Yaskawa INFORM job: X2_8A-21A(90,0)_HARDOX.JBI

/JOB
//NAME X2_8A-21A(90,0)_HARDOX
///FOLDERNAME X2
//POS
///NPOS 1752,1752,1752,46,0,0
///TOOL 0
///POSTYPE PULSE
///PULSE
C00000=-12667,-135547,-130714,31270,45596,0
C00001=-9315,-159766,-119262,-3212,6219,55552
C00002=-157761,-135547,-130714,31270,45596,-69143
C00003=-154472,-113934,-104337,41712,51336,-70449
C00004=-149832,-108771,-100172,39130,49259,-68869
C00005=-148058,-106656,-98467,38074,48499,-68236
C00006=-148062,-106275,-96666,38578,47777,-68578
C00007=-148058,-106656,-98467,38074,48499,-68236
C00008=-147997,-106381,-96958,38469,47847,-68508
C00009=-145894,-104035,-96109,36815,47477,-67498
C00010=-147997,-106381,-96958,38469,47847,-68508
C00011=-154410,-113635,-102825,42095,50721,-70729
C00012=-154342,-120637,-107041,25827,48602,-38771
C00013=-150292,-111683,-102360,22573,48994,-36710
C00014=-148798,-108210,-100464,21373,49171,-35962
C00015=-146664,-105787,-99597,19708,49308,-34937
C00016=-146949,-106220,-99797,19932,49282,-35074
C00017=-147721,-103636,-97533,20478,49410,-35405
C00018=-146949,-106220,-99797,19932,49282,-35074
C00019=-152261,-118724,-106469,24248,48548,-37770
C00020=-148295,-114597,-117137,-6490,60568,-69086
C00021=-147868,-109631,-111600,-6790,59752,-68875
C00022=-147704,-107727,-109395,-6911,59390,-68790
C00023=-147708,-107860,-107783,-6984,58336,-68724
C00024=-147704,-107727,-109395,-6911,59390,-68790
C00025=-147723,-107760,-107968,-6963,58499,-68740
C00026=-147306,-102596,-106094,-7098,60024,-68678
C00027=-147723,-107760,-107968,-6963,58499,-68740
C00028=-148315,-114751,-115749,-6537,59639,-69038
C00029=-148355,-114889,-117236,-6461,60467,-69101
C00030=-147925,-109892,-111692,-6763,59663,-68890
C00031=-147761,-107977,-109485,-6884,59305,-68805
C00032=-147764,-108104,-107870,-6957,58254,-68739
C00033=-147777,-108153,-108078,-6942,58354,-68751
C00034=-147358,-102980,-106206,-7078,59886,-68688
C00035=-147777,-108153,-108078,-6942,58354,-68751
C00036=-148373,-115211,-115873,-6515,59468,-69049
C00037=-147696,-122269,-111871,-35505,39043,-51945
C00038=-147690,-118447,-100224,-39719,34874,-49579
C00039=-148491,-109409,-94254,-38171,35277,-50420
C00040=-148787,-105724,-91002,-38010,35060,-50504
C00041=-148789,-105382,-89977,-38411,34697,-50285
C00042=-149058,-101689,-89016,-37046,35623,-51030
C00043=-149145,-100783,-88679,-36755,35795,-51189
C00044=-149058,-101689,-89016,-37046,35623,-51030
C00045=-145777,-99657,-88811,-39022,37803,-49998
C00046=-148139,-100407,-89095,-37251,36591,-50936
C00047=-145777,-99657,-88811,-39022,37803,-49998
C00048=-147690,-118447,-100224,-39719,34874,-49579
C00049=-128033,-128545,-103748,-39689,32513,-43973
C00050=-128383,-118409,-97778,-37905,33566,-44930
C00051=-128511,-114277,-94563,-37658,33626,-45064
C00052=-128512,-113804,-93446,-38069,33271,-44843
C00053=-129119,-111006,-93029,-36452,33958,-45715
C00054=-129434,-109852,-92636,-35862,34111,-46033
C00055=-128358,-113721,-93936,-37885,33613,-44941
C00056=-176216,-70111,-78093,55162,70856,-80763
C00057=-174311,-70781,-78417,54616,69674,-80426
C00058=-176216,-70111,-78093,55162,70856,-80763
C00059=-181747,-69996,-81392,56304,75271,-81045
C00060=-178033,-77165,-93769,42680,75059,-77098
C00061=-164745,-109340,-116699,-3009,62053,-68278
C00062=-145851,-112599,-102075,-47717,41998,-56322
C00063=-148044,-104803,-96379,-45883,41204,-57334
C00064=-148864,-101708,-93474,-45490,40644,-57533
C00065=-148866,-101457,-92299,-45986,40221,-57239
C00066=-148863,-101834,-94104,-45225,40876,-57690
C00067=-145127,-99228,-91361,-47944,42572,-56214
C00068=-147466,-100038,-91670,-46636,41186,-56907
C00069=-145127,-99228,-91361,-47944,42572,-56214
C00070=-146129,-107372,-95667,-48598,40993,-55782
C00071=-148216,-109089,-93488,-49289,38371,-55335
C00072=-148344,-107837,-93052,-48851,38553,-55585
C00073=-147906,-112054,-94498,-50363,37947,-54724
C00074=-145851,-112599,-102075,-47717,41998,-56322
C00075=-158250,-140903,-124067,-47621,67451,-49320
C00076=-161740,-133075,-117656,-46661,65672,-50232
C00077=-162335,-130592,-114553,-46699,64919,-50156
C00078=-162276,-129951,-113381,-46845,64676,-49998
C00079=-160420,-132544,-115533,-47350,65644,-49520
C00080=-135901,-74424,-73697,-74364,100921,-31256
C00081=-137788,-75503,-74147,-74218,99532,-31324
C00082=-138769,-76027,-74362,-74146,98812,-31363
C00083=-135901,-74424,-73697,-74364,100921,-31256
C00084=-149282,-147643,-98518,-79858,51263,-26133
C00085=-149394,-146891,-98381,-79629,51249,-26315
C00086=-148448,-152811,-99407,-81432,51428,-24854
C00087=-139735,-166147,-105854,-82069,56849,-22658
C00088=-180438,-97574,-115199,-33764,102267,52414
C00089=-189965,-108899,-115705,-31971,94091,51156
C00090=-189186,-107218,-114531,-32087,94499,51341
C00091=-189186,-107583,-113435,-32037,93763,51550
C00092=-190629,-109833,-115910,-31859,93547,51055
C00093=-186867,-102382,-113240,-32521,96788,51574
C00094=-187005,-102964,-110979,-32373,95300,51952
C00095=-188888,-106610,-112304,-32065,93703,51681
C00096=-187005,-102964,-110979,-32373,95300,51952
C00097=-188021,-107681,-112675,-32159,93748,52003
C00098=-189590,-103281,-111094,-32025,94271,51250
C00099=-188021,-107681,-112675,-32159,93748,52003
C00100=-180438,-97574,-115199,-33764,102267,52414
C00101=-185735,-83978,-109774,-33564,103394,50026
C00102=-199988,-77820,-108712,11582,98175,-38155
C00103=-204749,-56978,-92496,29836,109182,-47433
C00104=-202460,-56662,-91339,29422,107990,-46925
C00105=-201413,-57385,-91726,29256,107546,-46663
C00106=-201611,-57041,-91542,29296,107663,-46703
C00107=-201611,-58240,-90431,29070,106521,-47008
C00108=-203359,-50274,-87822,29763,109247,-46906
C00109=-195470,-25798,-72981,29209,109868,-43903
C00110=-195013,-27562,-73704,29036,109327,-43888
C00111=-194283,-28250,-74172,28893,109053,-43704
C00112=-194480,-28066,-74047,28932,109127,-43754
C00113=-194480,-29296,-73135,28708,108075,-44034
C00114=-195605,-24849,-71507,29147,109538,-44038
C00115=-191110,-5546,-57842,28597,109561,-42465
C00116=-192519,-3768,-54500,33008,111368,-41387
C00117=-191992,-5303,-55742,32912,111174,-41254
C00118=-192059,-5108,-55586,32924,111198,-41271
C00119=-192059,-6294,-54683,32651,110210,-41583
C00120=-192882,-2296,-53893,33162,111810,-41382
C00121=-203365,-15491,-64400,34648,115083,-44256
C00122=-218411,-26661,-75493,58573,107247,-46176
C00123=-145332,-87800,-123084,4045,108310,15756
C00124=-109199,-104290,-129101,-21867,105305,43874
C00125=-112610,-115777,-129409,-14908,94573,36374
C00126=-117115,-112620,-124614,-14006,92529,35127
C00127=-118008,-112320,-123068,-13816,91609,34934
C00128=-118007,-112900,-122267,-13806,90840,35020
C00129=-118044,-112536,-122505,-13803,91159,34973
C00130=-118576,-105776,-120168,-13731,93052,34586
C00131=-118044,-112536,-122505,-13803,91159,34973
C00132=-125955,-111499,-122045,-12179,90192,32457
C00133=-127333,-111877,-122174,-11884,89885,32033
C00134=-124755,-111115,-121914,-12435,90480,32824
C00135=-119624,-116552,-128230,-13509,92325,34321
C00136=-117231,-121833,-124467,-22052,85463,28755
C00137=-122341,-114124,-118662,-20866,84531,27121
C00138=-123318,-113111,-117155,-20643,83910,26885
C00139=-123641,-113323,-116249,-20585,83205,26892
C00140=-123595,-112804,-116375,-20585,83540,26851
C00141=-123397,-106736,-114247,-20589,85286,26623
C00142=-123595,-112804,-116375,-20585,83540,26851
C00143=-116023,-114044,-115764,-22346,84523,29358
C00144=-117346,-116777,-115957,-22098,82979,29171
C00145=-118867,-116723,-116143,-21757,82713,28674
C00146=-116293,-116772,-115815,-22329,83179,29512
C00147=-117231,-121833,-124467,-22052,85463,28755
C00148=-154726,-134692,-133300,19029,79240,32627
C00149=-155157,-123239,-125350,19102,80279,32639
C00150=-155214,-122106,-123677,19140,79867,32554
C00151=-155216,-122330,-122794,19175,79245,32454
C00152=-155272,-122641,-123186,19186,79334,32449
C00153=-154565,-115790,-120970,18882,81218,32994
C00154=-155272,-122449,-123985,19155,79894,32538
C00155=-110972,-119209,-121408,-15853,79302,48266
C00156=-109086,-133769,-122042,-16854,72857,49812
C00157=-111848,-135958,-122676,-16103,71595,48979
C00158=-109086,-133769,-122042,-16854,72857,49812
C00159=-108592,-130707,-130810,-16554,79646,49045
C00160=-120610,-122471,-119242,-21572,81234,22537
C00161=-120610,-122484,-118172,-21604,80613,22649
C00162=-120610,-122391,-116483,-21658,79689,22817
C00163=-120610,-122419,-116833,-21647,79876,22783
C00164=-120610,-122423,-116832,-21647,79874,22783
C00165=-120610,-122419,-116833,-21647,79876,22783
C00166=-120610,-122416,-116761,-21649,79836,22790
C00167=-120610,-122436,-116768,-21650,79830,22791
C00168=-120610,-122416,-116761,-21649,79836,22790
C00169=-120611,-122370,-120508,-21535,82009,22397
C00170=-120611,-120494,-126735,-3133,87635,4471
C00171=-120611,-121772,-123926,-3138,85252,4531
C00172=-120611,-122092,-122744,-3141,84362,4553
C00173=-120611,-122362,-121169,-3146,83256,4581
C00174=-120611,-122286,-121724,-3144,83636,4571
C00175=-120611,-122290,-121724,-3144,83633,4571
C00176=-120611,-122286,-121724,-3144,83636,4571
C00177=-120611,-121006,-125813,-3134,86805,4492
C00178=-120621,-120378,-125991,-12397,109990,35253
C00179=-136832,-143297,-133894,-19017,104291,40845
C00180=-187686,-122249,-118318,-34521,102174,42234
C00181=-187703,-122088,-115580,-34298,100833,42653
C00182=-187707,-122010,-114917,-34250,100525,42749
C00183=-187713,-121734,-113169,-34135,99743,42991
C00184=-187707,-122010,-114917,-34250,100525,42749
C00185=-187770,-121697,-112491,-32279,113674,44764
C00186=-187767,-121692,-112491,-32279,113678,44765
C00187=-187770,-121697,-112491,-32279,113674,44764
C00188=-187667,-121438,-112064,-34928,84963,41689
C00189=-187673,-121448,-112068,-34927,84958,41688
C00190=-187667,-121438,-112064,-34928,84963,41689
C00191=-187641,-121957,-115421,-34884,86463,41227
C00192=-173591,-141106,-131528,-9997,106250,69327
C00193=-160878,-120510,-126471,-37,121976,81968
C00194=-160881,-121699,-123664,-37,119637,81967
C00195=-160883,-121991,-122485,-37,118762,81967
C00196=-160886,-122244,-120905,-37,117660,81966
C00197=-160884,-122111,-121864,-37,118318,81967
C00198=-160882,-122100,-121862,-36,118322,81968
C00199=-160884,-122111,-121864,-37,118318,81967
C00200=-160879,-120821,-125908,-37,121469,81968
C00201=-160879,-120821,-131564,-37,121469,81968
C00202=-166129,-114439,-129167,13521,133132,-54375
C00203=-82387,-124374,-130385,21792,102809,-55833
C00204=-37550,-124758,-124791,27166,84975,-54517
C00205=-35933,-124831,-122904,26864,83389,-54284
C00206=-35589,-124875,-121597,26827,82538,-54351
C00207=-35584,-124889,-121174,26839,82296,-54405
C00208=-35764,-126387,-121953,26892,82093,-54519
C00209=-31633,-125451,-121673,25972,81076,-53208
C00210=-35764,-126387,-121953,26892,82093,-54519
C00211=-46981,-157328,-126723,35790,81436,-33730
C00212=-42905,-153934,-122174,35701,78867,-32870
C00213=-42758,-143813,-119569,35389,81762,-31868
C00214=-42905,-153934,-122174,35701,78867,-32870
C00215=-53188,-117519,-120731,36414,97747,-30962
C00216=-95179,-109851,-129540,3422,106316,17944
C00217=-143691,-100776,-119079,-26047,122130,73021
C00218=-146029,-112499,-120098,-24937,116556,73463
C00219=-147204,-116618,-119576,-24569,113992,73590
C00220=-147487,-116577,-118677,-24502,113425,73607
C00221=-146967,-116625,-120319,-24630,114475,73574
C00222=-147345,-121113,-121824,-24401,113105,73737
C00223=-146899,-128254,-123879,-23878,111030,74376
C00224=-147345,-121113,-121824,-24401,113105,73737
C00225=-118081,-135478,-120686,-30293,109901,65237
C00226=-118366,-136707,-118609,-29972,108136,65614
C00227=-120887,-140213,-119894,-30302,106351,65070
C00228=-118366,-136707,-118609,-29972,108136,65614
C00229=-117820,-130449,-123242,-31209,113594,64262
C00230=-93926,-103398,-125362,-18301,106221,39936
C00231=-72688,-110808,-124077,-7134,85250,24096
C00232=-75848,-101444,-116923,-6191,85411,23073
C00233=-76170,-100985,-115528,-6097,84767,23002
C00234=-76167,-101481,-114835,-6104,84090,23035
C00235=-78739,-96930,-113773,-5320,85595,22140
C00236=-79843,-95445,-113201,-4985,85938,21775
C00237=-77748,-98228,-114268,-5620,85298,22470
C00238=-140085,-104632,-109249,40944,98797,-6712
C00239=-140263,-103640,-106572,40817,98007,-7102
C00240=-137942,-102173,-106029,40697,97269,-6378
C00241=-140263,-103640,-106572,40817,98007,-7102
C00242=-135988,-101428,-112112,41019,99549,-4631
C00243=-141957,-83285,-117139,12315,91699,6710
C00244=-161957,-129781,-122866,-20018,67926,12328
C00245=-166016,-109699,-113650,-17211,72980,10098
C00246=-166795,-105246,-111748,-16434,74862,9605
C00247=-165677,-113012,-111900,-18316,68836,10778
C00248=-162725,-116093,-113629,-19548,69016,11850
C00249=-162651,-107484,-110669,-19284,71494,11460
C00250=-162725,-116093,-113629,-19548,69016,11850
C00251=-155151,-112727,-112486,-22270,71877,14160
C00252=-155120,-113819,-110277,-22518,70103,14518
C00253=-159000,-114269,-110433,-21107,68960,13264
C00254=-155120,-113819,-110277,-22518,70103,14518
C00255=-155137,-138999,-124748,-23105,66364,15269
C00256=-81055,-115973,-127517,23586,109336,-64560
C00257=-76492,-127739,-126040,22738,101683,-64421
C00258=-76072,-128597,-125529,22671,100870,-64425
C00259=-76065,-128640,-125326,22657,100732,-64448
C00260=-76072,-128576,-125785,22685,101025,-64394
C00261=-82641,-146978,-130130,22016,96499,-67668
C00262=-81130,-155003,-132256,21951,93476,-67670
C00263=-82641,-146978,-130130,22016,96499,-67668
C00264=-84000,-144678,-127518,21929,96467,-68175
C00265=-84000,-143983,-126065,21900,95967,-68269
C00266=-83327,-146231,-127404,21916,95478,-68108
C00267=-88356,-135439,-132684,22407,104994,-68175
C00268=-104080,-128245,-132212,-31995,84146,-22143
C00269=-106783,-105266,-117364,-31197,85468,-23533
C00270=-107129,-103609,-115494,-31111,85090,-23558
C00271=-107127,-104217,-114421,-31144,84251,-23329
C00272=-107044,-104571,-114816,-31164,84333,-23320
C00273=-107880,-99055,-112779,-30885,85404,-23924
C00274=-107044,-104571,-114816,-31164,84333,-23320
C00275=-105114,-115284,-123193,-31689,84721,-22698
C00276=-105208,-113465,-123990,-31624,85910,-23065
C00277=-106823,-104635,-117017,-31184,85549,-23570
C00278=-107122,-103295,-115264,-31113,85109,-23561
C00279=-107121,-103855,-114286,-31142,84342,-23351
C00280=-107087,-104437,-114776,-31151,84356,-23343
C00281=-107921,-98925,-112738,-30873,85426,-23945
C00282=-107087,-104437,-114776,-31151,84356,-23343
C00283=-105701,-116384,-125830,-31502,85418,-23114
C00284=-79137,-116524,-127291,-7118,77084,38210
C00285=-66518,-158449,-133200,-8588,59166,50817
C00286=-70166,-147728,-127011,-6864,60501,49298
C00287=-71549,-143558,-123868,-6244,60595,48757
C00288=-71544,-142942,-122687,-6271,60188,48782
C00289=-71412,-140542,-122600,-6259,61371,48766
C00290=-74130,-137647,-121783,-5023,62161,47690
C00291=-71412,-140542,-122600,-6259,61371,48766
C00292=-59221,-85077,-106862,-19044,97138,55247
C00293=-59772,-90133,-108950,-18878,95774,55276
C00294=-59221,-85077,-106862,-19044,97138,55247
C00295=-65406,-128676,-128270,-8670,80773,42177
C00296=-57064,-112054,-129147,-2862,108793,29097
C00297=-70948,-123089,-127271,10962,111372,-380
C00298=-67644,-116564,-123033,11394,111660,848
C00299=-67644,-116773,-122597,11361,111292,811
C00300=-67644,-116291,-123546,11437,112109,893
C00301=-70770,-123262,-125779,10903,110357,-412
C00302=-70770,-123588,-124717,10837,109552,-488
C00303=-69306,-120453,-123728,11077,110342,115
C00304=-70770,-123283,-125719,10898,110311,-416
C00305=-70770,-119886,-130778,11344,115083,53
C00306=-68413,-122856,-123349,22437,117236,58
C00307=-67404,-122631,-120786,22344,115611,123
C00308=-67401,-122683,-120099,22253,115193,37
C00309=-67283,-122594,-120333,22317,115338,115
C00310=-65261,-118175,-118917,23034,116088,1096
C00311=-67283,-122594,-120333,22317,115338,115
C00312=-70820,-123560,-126018,22187,119059,-540
C00313=-59587,-128850,-129971,-18356,103459,48793
C00314=-60648,-112549,-116046,-37363,97913,74718
C00315=-66648,-121539,-115269,-36526,91263,74498
C00316=-69624,-125916,-115212,-36242,88151,74300
C00317=-69624,-125773,-114639,-36242,87924,74374
C00318=-69624,-125814,-114800,-36242,87987,74354
C00319=-70738,-127677,-115368,-36152,87024,74211
C00320=-69624,-125814,-114800,-36242,87987,74354
C00321=-61556,-115340,-115782,-37136,96245,74919
C00322=-93863,-107857,-129738,-18786,98098,27923
C00323=-113340,-105978,-120535,-17383,92037,15860
C00324=-116256,-99504,-115214,-16745,91512,14962
C00325=-117355,-97038,-113094,-16498,91266,14630
C00326=-124053,-106600,-116618,-14934,87391,12894
C00327=-123019,-109757,-118902,-15179,87365,13243
C00328=-120254,-118381,-124729,-15823,87055,14212
C00329=-121076,-118719,-112405,-41381,81563,9211
C00330=-125328,-110839,-107644,-40465,80446,7775
C00331=-126920,-107772,-105722,-40091,80023,7243
C00332=-122279,-105715,-102241,-45382,81605,7865
C00333=-118123,-103314,-98388,-50429,83325,8212
C00334=-115452,-99808,-95169,-50805,84680,8860
C00335=-113598,-101964,-96694,-51043,85596,9323
C00336=-108732,-107177,-100380,-51565,88044,10518
C00337=-131658,-113091,-133069,-11905,90618,-13395
C00338=-155934,-143784,-122811,23124,58745,-32427
C00339=-151507,-132468,-117411,20635,59886,-30339
C00340=-149876,-128251,-115276,19729,60288,-29596
C00341=-151213,-128323,-114307,20456,60014,-30191
C00342=-146890,-120795,-114089,13688,65901,-25886
C00343=-142734,-111238,-112703,7950,73001,-22079
C00344=-143750,-114926,-115045,8343,72653,-22456
C00345=-146492,-125018,-121022,9420,71459,-23506
C00346=-146459,-122334,-129315,9145,77857,-23007
C00347=-118526,-115013,-133262,8809,105739,-46794
C00348=-93674,-118800,-129721,8134,120991,-68616
C00349=-93669,-120967,-127104,7892,118292,-68817
C00350=-93667,-121558,-126026,7814,117333,-68886
C00351=-93663,-121536,-126144,7822,117416,-68879
C00352=-93639,-121762,-126135,7818,117296,-68878
C00353=-93680,-121434,-126040,7817,117406,-68885
C00354=-93660,-121042,-127131,7893,118270,-68815
C00355=-93665,-118880,-129750,8134,120967,-68614
C00356=-98446,-113408,-116165,41475,93741,-73013
C00357=-93996,-117843,-114815,40802,89312,-72817
C00358=-91343,-117266,-113836,40455,87860,-72224
C00359=-92137,-119395,-114109,40564,87510,-72703
C00360=-95072,-126184,-113786,40951,86041,-74561
C00361=-95071,-125918,-112907,40977,85731,-74679
C00362=-96936,-125131,-114749,41104,87782,-74702
C00363=-101504,-121000,-116278,41571,92256,-74948
C00364=-100864,-122088,-112493,43204,76282,-71688
C00365=-95643,-121963,-109784,42340,72556,-70846
C00366=-93677,-120964,-108398,41948,71358,-70433
C00367=-93599,-121011,-107366,42074,70823,-70622
C00368=-95642,-121622,-108630,42447,72155,-71017
C00369=-100864,-121830,-111367,43291,75868,-71867
C00370=-131033,-115476,-133015,2815,101744,-74384
C00371=-151471,-119125,-123137,-34971,103386,-73225
C00372=-162012,-101235,-114016,-37763,108592,-75954
C00373=-163593,-104354,-113811,-37340,106547,-75879
C00374=-162938,-104376,-113793,-37349,106803,-75692
C00375=-158829,-104862,-111593,-37019,107224,-74083
C00376=-157962,-101866,-111865,-37402,108959,-74341
C00377=-155898,-93647,-112180,-38609,113341,-75115
C00378=-179206,-139250,-107986,-62075,77828,-66561
C00379=-185232,-138953,-105140,-62379,73225,-66913
C00380=-187696,-139015,-104542,-62453,71468,-67163
C00381=-187702,-137665,-102648,-62587,71237,-66963
C00382=-185238,-138055,-103864,-62461,73065,-66778
C00383=-179211,-138396,-106727,-62132,77661,-66424
C00384=-179188,-148562,-121526,-61524,79591,-68010
C00385=-184417,-115822,-131978,-19629,107310,7500
C00386=-190427,-134899,-136820,8574,116374,78562
C00387=-188066,-120573,-128029,9218,118052,79593
C00388=-191610,-147357,-136376,6897,103791,75181
C00389=-187795,-119828,-126345,9210,117376,79639
C00390=-187841,-121664,-124728,-2971,114560,78170
C00391=-187942,-121398,-126015,-3016,115485,78109
C00392=-187937,-119495,-128851,-3098,118205,78035
C00393=-176042,-128909,-129640,-7380,110692,58022
C00394=-187833,-113452,-115854,-34994,105139,41767
C00395=-187847,-113781,-113588,-34722,103839,42187
C00396=-187853,-113844,-112659,-34623,103335,42348
C00397=-187856,-113866,-111596,-34519,102780,42525
C00398=-187851,-113844,-112538,-34611,103274,42368
C00399=-187836,-113627,-114840,-34866,104547,41960
C00400=-186756,-108501,-120882,-36201,110201,40487
C00401=-150585,-129060,-123753,-46684,114085,-39870
C00402=-134046,-137019,-115206,-49635,112096,-74674
C00403=-134033,-140586,-110307,-48065,108843,-72866
C00404=-134037,-138671,-107458,-47843,108316,-72589
C00405=-133950,-137111,-106105,-47812,108341,-72556
C00406=-133930,-150358,-126108,1173,113974,-57522
C00407=-133955,-150680,-126140,1162,113827,-57532
C00408=-134042,-144068,-115274,40466,90158,-47055
C00409=-134072,-145102,-116392,40468,90292,-47016
C00410=-134074,-146851,-118858,40485,90771,-46834
C00411=-141855,-151854,-132376,33568,89282,-32323
C00412=-173958,-148748,-133240,11874,65312,15203
C00413=-187653,-128002,-123664,-7056,57779,46476
C00414=-188071,-112180,-99768,1790,31671,46486
C00415=-188092,-111455,-97340,1875,30550,46442
C00416=-187851,-111485,-96835,1581,30220,46589
C00417=-187792,-110201,-93997,1555,29133,46605
C00418=-187737,-110060,-93474,1490,28882,46636
C00419=-187785,-109075,-90961,1604,27844,46576
C00420=-188106,-109627,-92159,2030,28303,46362
C00421=-188086,-110531,-94662,1935,29378,46411
C00422=-188086,-114129,-114927,1479,39995,46659
C00423=-201470,-41376,-102585,19941,97743,-57993
C00424=-197439,-2624,-49840,39121,107911,-51008
C00425=-168348,92819,48556,27514,116832,-48709
C00426=-170146,82769,36005,28011,119675,-48673
C00427=-172466,59662,8523,30747,114377,-38085
C00428=-173361,44293,-8668,31536,116980,-37634
C00429=-173326,42548,-10417,31798,119739,-39927
C00430=-173293,31446,-22173,31559,124382,-42741
C00431=-170045,43132,-9775,28753,130915,-51393
C00432=-186843,33187,-28183,45340,118495,-56566
C00433=-187270,22965,-40018,42118,113549,-44205
C00434=-164927,12374,-50848,37497,97302,26684
C00435=-160848,-52651,-98971,6904,73590,44156
C00436=-187933,-111679,-98706,-278,30585,46526
C00437=-187953,-110958,-96368,-260,29517,46517
C00438=-188171,-110591,-95666,34,29272,46369
C00439=-188111,-109885,-93130,-50,28074,46412
C00440=-188090,-109778,-92606,-82,27808,46427
C00441=-188055,-108797,-90194,-133,26826,46455
C00442=-187968,-109087,-91174,-258,27282,46516
C00443=-187948,-109974,-93584,-278,28309,46526
C00444=-190713,-138118,-122139,3147,45685,54861
C00445=-188097,-104568,-127563,3199,90457,72619
C00446=-188112,-108983,-124849,3203,86524,72515
C00447=-196049,-130715,-128058,11352,73875,69900
C00448=-193131,-119078,-125609,7963,80164,71095
C00449=-187364,-124777,-127140,2732,76642,72458
C00450=-191510,-130298,-128202,6704,73471,71168
C00451=-188153,-109076,-124888,3215,86502,72501
C00452=-188138,-104664,-127604,3212,90434,72606
C00453=-187898,-111965,-120493,-16766,69565,69566
C00454=-187918,-113285,-117348,-17044,67055,69927
C00455=-188336,-115132,-116370,-17036,65483,70009
C00456=-188181,-112945,-115606,-17029,66143,69965
C00457=-188166,-113080,-115592,-17048,66072,69982
C00458=-187991,-112297,-115306,-17102,66325,70009
C00459=-187944,-113344,-117352,-17035,67023,69922
C00460=-187924,-112030,-120500,-16757,69531,69561
C00461=-180038,-109975,-126789,-2440,82512,-7441
C00462=-174468,-102021,-118148,-1871,82653,-17547
C00463=-174479,-103807,-115834,-1877,80312,-17516
C00464=-175021,-104384,-114967,-1695,79470,-17680
C00465=-174783,-104250,-115053,-1777,79597,-17606
C00466=-174170,-106690,-109656,-11758,69864,-18312
C00467=-172833,-107431,-109671,-12341,69693,-17819
C00468=-174390,-105691,-110273,-11607,70709,-18474
C00469=-174377,-104937,-112785,-11492,72607,-18653
C00470=-190845,-100837,-124447,13698,93294,-33124
C00471=-206306,-116062,-120388,37359,88631,-50073
C00472=-215039,-120395,-106715,50971,83253,-62053
C00473=-215038,-119729,-104733,51036,82687,-62365
C00474=-215037,-119445,-103934,51064,82464,-62488
C00475=-215047,-118488,-101366,51160,81769,-62880
C00476=-215047,-118800,-102176,51129,81987,-62759
C00477=-215049,-119543,-104187,51057,82539,-62453
C00478=-215012,-122438,-115563,50746,86080,-60488
C00479=-160845,-113405,-113287,47121,77099,31472
C00480=-160851,-113463,-110064,47446,75709,30781
C00481=-161282,-114943,-109409,47754,75135,30277
C00482=-161254,-114846,-109376,47745,75139,30294
C00483=-160788,-113231,-109982,47419,75724,30819
C00484=-160782,-112987,-114684,46949,77813,31850
C00485=-161690,-87231,-108001,36248,90547,80444
C00486=-156210,-91223,-102127,34873,83736,80390
C00487=-152348,-73560,-94415,33644,85868,82536
C00488=-158330,-83683,-104653,35339,89043,81248
C00489=-160758,-112853,-114863,36163,82877,78288
C00490=-160760,-113152,-111426,36317,81029,77674
C00491=-159491,-108015,-113138,31549,97627,78488
C00492=-160662,-113202,-114930,31505,96709,77777
C00493=-163626,-124672,-119545,29271,98661,76908
C00494=-164622,-129006,-121133,28240,99357,76613
C00495=-160757,-112482,-116558,30024,102576,77779
C00496=-160755,-111254,-119690,30396,104801,78387
C00497=-139139,-104942,-132434,5076,105021,81413
C00498=-120610,-140892,-128239,-26796,83300,73925
C00499=-124485,-139346,-124335,-26282,80622,73071
C00500=-128794,-174695,-130569,-28116,58521,76693
C00501=-123854,-173705,-127920,-33486,56775,79744
C00502=-127596,-155142,-123084,-28725,56836,77726
C00503=-128095,-155529,-122172,-29132,53686,78388
C00504=-128860,-155984,-126780,-25446,58633,74277
C00505=-138109,-135032,-133743,-8289,74304,51513
C00506=-203654,-125968,-124215,37381,73551,-30645
C00507=-201127,-103516,-110680,20461,62884,-59060
C00508=-201138,-104157,-107983,20829,61019,-59420
C00509=-201193,-104400,-106652,21043,60147,-59612
C00510=-201232,-104446,-106694,21063,60161,-59627
C00511=-200873,-105228,-106882,20926,59802,-59552
C00512=-201116,-104130,-107973,20816,61021,-59411
C00513=-201105,-103488,-110669,20449,62886,-59051
C00514=-198523,-119273,-121454,24683,77158,-64296
C00515=-174403,-100049,-121231,21877,99309,-62114
C00516=-174406,-102879,-118773,21681,96545,-62622
C00517=-172958,-103152,-117900,21399,95556,-62302
C00518=-174224,-104881,-115910,21520,93897,-63036
C00519=-174418,-104205,-117181,21599,94999,-62906
C00520=-174415,-101880,-119808,21752,97619,-62429
C00521=-185776,-93152,-118465,-1785,83350,-67432
C00522=-169060,-142396,-123848,-37084,49654,-60484
C00523=-174230,-113472,-108308,-34615,49911,-64397
C00524=-174247,-112967,-104740,-35556,48304,-63744
C00525=-174471,-112928,-103062,-35946,47380,-63468
C00526=-174489,-112275,-102294,-36008,47261,-63425
C00527=-174590,-112153,-101603,-36140,46922,-63333
C00528=-174396,-113097,-100663,-36857,46141,-62871
C00529=-174330,-114043,-100633,-37190,45762,-62656
C00530=-174129,-122060,-98220,-45554,37107,-60115
C00531=-174246,-112406,-102200,-36228,47262,-63291
C00532=-174229,-113129,-105847,-35265,48804,-63944
C00533=-182962,-136134,-123657,-29797,44727,-67038
C00534=-210827,-121899,-127370,-35396,86436,-76908
C00535=-214505,-124636,-123608,-35577,86411,-76994
C00536=-214521,-124823,-120077,-35640,84542,-76397
C00537=-209595,-138372,-118962,-40572,76618,-76704
C00538=-215572,-134536,-117924,-37557,71164,-81051
C00539=-214545,-124844,-120083,-35636,84527,-76402
C00540=-214528,-124659,-123615,-35573,86395,-76999
C00541=-214596,-124890,-121786,-39550,96156,-78039
C00542=-214607,-124784,-118461,-39383,94595,-77461
C00543=-215336,-122839,-115954,-39308,93846,-77495
C00544=-215216,-123286,-113688,-39218,92622,-76995
C00545=-214785,-119888,-114308,-39371,94481,-77497
C00546=-214619,-124823,-118761,-39395,94718,-77513
C00547=-214540,-124430,-116246,-48349,86426,-68042
C00548=-214499,-123956,-126099,-48385,90728,-70182
C00549=-158797,-145907,-128305,-56145,74291,-56792
C00550=-118138,-117595,-113507,-59219,64127,-52420
C00551=-134091,-119062,-102284,-58108,50235,-52331
C00552=-134095,-117716,-98836,-59129,49460,-51612
C00553=-134657,-117185,-97454,-59366,48806,-51448
C00554=-134083,-121591,-110246,-11584,43366,-62365
C00555=-133895,-121523,-110170,-11744,43379,-62274
C00556=-133843,-121378,-109751,-11603,42967,-62923
C00557=-134088,-120272,-105685,-8075,39028,-71413
C00558=-134097,-120880,-107281,-7954,39689,-71484
C00559=-133538,-122024,-122159,-7272,48238,-71950
C00560=-134045,-120979,-109361,-39707,45136,-55893
C00561=-134048,-117179,-98466,-43015,41514,-53843
C00562=-133905,-117568,-98535,-40781,40764,-54269
C00563=-134181,-118830,-102497,-12918,37668,-61575
C00564=-134087,-119212,-102754,-13019,37648,-61516
C00565=-123717,-118705,-98316,36301,38159,-75512
C00566=-134076,-115553,-94209,55177,43841,-79182
C00567=-133651,-114033,-99266,51853,45977,-77066
C00568=-134816,-132236,-131789,-6177,48808,-72548
C00569=-152519,-98596,-126841,-17039,86437,-59409
C00570=-167034,-82548,-116958,-26153,108191,-47353
C00571=-167227,-85698,-113927,-25595,104988,-46679
C00572=-154754,-79329,-105712,-37422,108521,-45283
C00573=-159285,-74428,-103512,-37136,107681,-46815
C00574=-167896,-62467,-97746,-36329,106502,-49789
C00575=-170836,-57718,-95291,-35960,106173,-50801
C00576=-180979,-58723,-101497,-23976,107062,-51805
C00577=-180909,-54943,-104050,-24554,110296,-52487
C00578=-168157,-75412,-102271,-33648,91006,-21456
C00579=-174012,-67106,-91297,-33471,82630,-14810
C00580=-175466,-61382,-85667,-32996,81659,-15067
C00581=-176013,-59150,-83405,-32819,81253,-15153
C00582=-202608,-62025,-89962,4221,78254,-36710
C00583=-159972,-87195,-101610,-14286,75081,-22762
C00584=-154310,-93015,-102157,-19304,70769,-24486
C00585=-154362,-96202,-104591,-19297,70625,-24481
C00586=-154503,-104813,-110762,-19306,69999,-24428
C00587=-155575,-73729,-96860,-32555,86012,-14938
C00588=-157088,-68154,-91284,-32096,84992,-15206
C00589=-157731,-66276,-89193,-31903,84490,-15302
C00590=-176839,-77218,-97385,-7105,75561,-28432
C00591=-165473,-80321,-98709,-11948,76053,-24715
C00592=-199796,-81518,-91231,35244,71315,-57262
C00593=-201423,-82172,-92479,35779,72324,-57601
C00594=-205660,-83542,-95477,37134,74990,-58446
C00595=-150225,-90058,-124320,-20069,81923,-14603
C00596=-88917,-116100,-126028,-29630,66347,39612
C00597=-48102,-114880,-112674,-35477,56596,75725
C00598=-53396,-105773,-101201,-33500,52497,74682
C00599=-53385,-105323,-98106,-34230,51099,75219
C00600=-48465,-101460,-95464,-40425,56724,79171
C00601=-72122,-108844,-98440,461,39847,55622
C00602=-53363,-105522,-99057,-19217,46878,60217
C00603=-53371,-105892,-101942,-18746,48378,59901
C00604=-53322,-113038,-104699,812,43724,42660
C00605=-53318,-112442,-102021,830,42382,42650
C00606=-53317,-112163,-100935,837,41857,42645
C00607=-53253,-112229,-97736,1547,37461,42516
C00608=-53300,-111445,-98358,1568,38246,42506
C00609=-51520,-115460,-104005,-179,39644,43460
C00610=-55761,-139961,-122674,-27476,66843,55729
C00611=-53542,-121644,-113892,-40363,83761,61539
C00612=-53523,-121175,-111327,-40444,82737,61941
C00613=-53533,-120846,-110023,-41635,87424,59647
C00614=-53533,-120798,-109834,-41636,87355,59676
C00615=-53529,-120315,-108043,-41648,86710,59935
C00616=-53536,-120580,-109029,-41640,87063,59791
C00617=-53556,-121151,-111460,-41628,87965,59422
C00618=-52633,-122748,-126719,-40391,89833,59612
C00619=-140119,-108661,-130674,-21165,82789,-25459
C00620=-161125,-123349,-120158,-18581,66270,-46079
C00621=-161135,-123185,-116439,-18891,64175,-45732
C00622=-161140,-122976,-114905,-19018,63381,-45597
C00623=-161216,-123269,-115002,-18998,63277,-45609
C00624=-162856,-121662,-114495,-18189,63396,-46272
C00625=-161212,-123488,-116538,-18871,64068,-45743
C00626=-161202,-123677,-120265,-18562,66156,-46089
C00627=-167124,-146469,-125858,32695,63076,-70922
C00628=-161220,-122264,-110536,44525,64077,-74742
C00629=-161219,-121375,-107584,44985,63095,-75224
C00630=-164956,-113855,-102560,48427,66781,-75111
C00631=-161213,-120936,-106323,43985,60856,-74418
C00632=-161480,-119492,-104017,44742,56174,-74995
C00633=-161477,-119788,-101535,47560,52624,-77093
C00634=-161197,-119682,-102993,46927,53134,-76618
C00635=-161197,-120736,-105876,46275,53998,-76117
C00636=-161177,-121556,-108554,35078,57327,-43050
C00637=-161177,-120932,-106617,35398,56609,-43319
C00638=-152937,-127654,-109782,25136,48983,-42100
C00639=-161176,-119640,-103030,36318,54707,-44163
C00640=-161179,-121241,-107541,34339,64662,-45277
C00641=-161179,-121533,-108462,34233,65010,-45160
C00642=-161180,-122193,-110741,33972,65899,-44866
C00643=-159909,-111206,-128347,-10927,59798,-43136
C00644=-174276,-119239,-128019,9099,73009,32604
C00645=-174287,-122281,-118814,9519,65873,32039
C00646=-174304,-122135,-115653,9666,64029,31878
C00647=-174310,-121974,-114355,9727,63324,31815
C00648=-174277,-122172,-120616,-9764,82080,37769
C00649=-174277,-122177,-120568,-9764,82048,37772
C00650=-174317,-121775,-113110,-33515,107538,43031
C00651=-174312,-121937,-114098,-33622,107981,42892
C00652=-174299,-122214,-116525,-33911,109120,42531
C00653=-174287,-119835,-127268,-36019,115609,40290
C00654=-15972,-110889,-128286,-10965,59905,-43045
C00655=-12667,-135547,-130714,31270,45596,0
C00656=-9315,-159766,-119262,-3212,6219,55552
C00657=-157761,-135547,-130714,31270,45596,-69143
C00658=-154472,-113934,-104337,41712,51336,-70449
C00659=-149832,-108771,-100172,39130,49259,-68869
C00660=-148058,-106656,-98467,38074,48499,-68236
C00661=-148062,-106275,-96666,38578,47777,-68578
C00662=-148058,-106656,-98467,38074,48499,-68236
C00663=-147997,-106381,-96958,38469,47847,-68508
C00664=-145894,-104035,-96109,36815,47477,-67498
C00665=-147997,-106381,-96958,38469,47847,-68508
C00666=-154410,-113635,-102825,42095,50721,-70729
C00667=-154342,-120637,-107041,25827,48602,-38771
C00668=-150292,-111683,-102360,22573,48994,-36710
C00669=-148798,-108210,-100464,21373,49171,-35962
C00670=-146664,-105787,-99597,19708,49308,-34937
C00671=-146949,-106220,-99797,19932,49282,-35074
C00672=-147721,-103636,-97533,20478,49410,-35405
C00673=-146949,-106220,-99797,19932,49282,-35074
C00674=-152261,-118724,-106469,24248,48548,-37770
C00675=-148295,-114597,-117137,-6490,60568,-69086
C00676=-147868,-109631,-111600,-6790,59752,-68875
C00677=-117093,-120499,-115228,-23648,62285,-57221
C00678=-113886,-102168,-107256,-24278,67338,-57062
C00679=-113886,-102375,-106001,-24426,66534,-56885
C00680=-113886,-102359,-106115,-24413,66607,-56901
C00681=-113886,-102359,-106115,-24413,66607,-56901
C00682=-114646,-97769,-104385,-23859,67577,-57404
C00683=-114475,-101992,-107821,-23944,67574,-57337
C00684=-147704,-107727,-109395,-6911,59390,-68790
C00685=-147708,-107860,-107783,-6984,58336,-68724
C00686=-147704,-107727,-109395,-6911,59390,-68790
C00687=-147723,-107760,-107968,-6963,58499,-68740
C00688=-147306,-102596,-106094,-7098,60024,-68678
C00689=-147723,-107760,-107968,-6963,58499,-68740
C00690=-148315,-114751,-115749,-6537,59639,-69038
C00691=-148355,-114889,-117236,-6461,60467,-69101
C00692=-147925,-109892,-111692,-6763,59663,-68890
C00693=-147761,-107977,-109485,-6884,59305,-68805
C00694=-147764,-108104,-107870,-6957,58254,-68739
C00695=-147777,-108153,-108078,-6942,58354,-68751
C00696=-147358,-102980,-106206,-7078,59886,-68688
C00697=-147777,-108153,-108078,-6942,58354,-68751
C00698=-148373,-115211,-115873,-6515,59468,-69049
C00699=-147696,-122269,-111871,-35505,39043,-51945
C00700=-147690,-118447,-100224,-39719,34874,-49579
C00701=-148491,-109409,-94254,-38171,35277,-50420
C00702=-148787,-105724,-91002,-38010,35060,-50504
C00703=-148789,-105382,-89977,-38411,34697,-50285
C00704=-149058,-101689,-89016,-37046,35623,-51030
C00705=-149145,-100783,-88679,-36755,35795,-51189
C00706=-149058,-101689,-89016,-37046,35623,-51030
C00707=-145777,-99657,-88811,-39022,37803,-49998
C00708=-148139,-100407,-89095,-37251,36591,-50936
C00709=-145777,-99657,-88811,-39022,37803,-49998
C00710=-147690,-118447,-100224,-39719,34874,-49579
C00711=-128033,-128545,-103748,-39689,32513,-43973
C00712=-128383,-118409,-97778,-37905,33566,-44930
C00713=-128511,-114277,-94563,-37658,33626,-45064
C00714=-128512,-113804,-93446,-38069,33271,-44843
C00715=-129119,-111006,-93029,-36452,33958,-45715
C00716=-129434,-109852,-92636,-35862,34111,-46033
C00717=-128358,-113721,-93936,-37885,33613,-44941
C00718=-176216,-70111,-78093,55162,70856,-80763
C00719=-174311,-70781,-78417,54616,69674,-80426
C00720=-176216,-70111,-78093,55162,70856,-80763
C00721=-181747,-69996,-81392,56304,75271,-81045
C00722=-178033,-77165,-93769,42680,75059,-77098
C00723=-164745,-109340,-116699,-3009,62053,-68278
C00724=-145851,-112599,-102075,-47717,41998,-56322
C00725=-148044,-104803,-96379,-45883,41204,-57334
C00726=-148864,-101708,-93474,-45490,40644,-57533
C00727=-148866,-101457,-92299,-45986,40221,-57239
C00728=-148863,-101834,-94104,-45225,40876,-57690
C00729=-145127,-99228,-91361,-47944,42572,-56214
C00730=-147466,-100038,-91670,-46636,41186,-56907
C00731=-145127,-99228,-91361,-47944,42572,-56214
C00732=-146129,-107372,-95667,-48598,40993,-55782
C00733=-148216,-109089,-93488,-49289,38371,-55335
C00734=-148344,-107837,-93052,-48851,38553,-55585
C00735=-147906,-112054,-94498,-50363,37947,-54724
C00736=-145851,-112599,-102075,-47717,41998,-56322
C00737=-158250,-140903,-124067,-47621,67451,-49320
C00738=-161740,-133075,-117656,-46661,65672,-50232
C00739=-162335,-130592,-114553,-46699,64919,-50156
C00740=-162276,-129951,-113381,-46845,64676,-49998
C00741=-160420,-132544,-115533,-47350,65644,-49520
C00742=-135901,-74424,-73697,-74364,100921,-31256
C00743=-137788,-75503,-74147,-74218,99532,-31324
C00744=-138769,-76027,-74362,-74146,98812,-31363
C00745=-135901,-74424,-73697,-74364,100921,-31256
C00746=-149282,-147643,-98518,-79858,51263,-26133
C00747=-149394,-146891,-98381,-79629,51249,-26315
C00748=-148448,-152811,-99407,-81432,51428,-24854
C00749=-139735,-166147,-105854,-82069,56849,-22658
C00750=-180438,-97574,-115199,-33764,102267,52414
C00751=-189965,-108899,-115705,-31971,94091,51156
C00752=-190633,-110068,-115194,-31831,93066,51189
C00753=-190637,-110288,-114404,-31804,92551,51332
C00754=-190629,-109833,-115910,-31859,93547,51055
C00755=-186867,-102382,-113240,-32521,96788,51574
C00756=-187005,-102964,-110979,-32373,95300,51952
C00757=-188888,-106610,-112304,-32065,93703,51681
C00758=-187005,-102964,-110979,-32373,95300,51952
C00759=-188021,-107681,-112675,-32159,93748,52003
C00760=-189590,-103281,-111094,-32025,94271,51250
C00761=-188021,-107681,-112675,-32159,93748,52003
C00762=-180438,-97574,-115199,-33764,102267,52414
C00763=-185735,-83978,-109774,-33564,103394,50026
C00764=-199988,-77820,-108712,11582,98175,-38155
C00765=-204749,-56978,-92496,29836,109182,-47433
C00766=-202460,-56662,-91339,29422,107990,-46925
C00767=-201413,-57385,-91726,29256,107546,-46663
C00768=-201611,-57041,-91542,29296,107663,-46703
C00769=-201611,-58240,-90431,29070,106521,-47008
C00770=-203359,-50274,-87822,29763,109247,-46906
C00771=-195470,-25798,-72981,29209,109868,-43903
C00772=-195013,-27562,-73704,29036,109327,-43888
C00773=-194283,-28250,-74172,28893,109053,-43704
C00774=-194480,-28066,-74047,28932,109127,-43754
C00775=-194480,-29296,-73135,28708,108075,-44034
C00776=-195605,-24849,-71507,29147,109538,-44038
C00777=-191110,-5546,-57842,28597,109561,-42465
C00778=-192519,-3768,-54500,33008,111368,-41387
C00779=-191992,-5303,-55742,32912,111174,-41254
C00780=-192059,-5108,-55586,32924,111198,-41271
C00781=-192059,-6294,-54683,32651,110210,-41583
C00782=-192882,-2296,-53893,33162,111810,-41382
C00783=-203365,-15491,-64400,34648,115083,-44256
C00784=-218411,-26661,-75493,58573,107247,-46176
C00785=-145332,-87800,-123084,4045,108310,15756
C00786=-109199,-104290,-129101,-21867,105305,43874
C00787=-112610,-115777,-129409,-14908,94573,36374
C00788=-117115,-112620,-124614,-14006,92529,35127
C00789=-118008,-112320,-123068,-13816,91609,34934
C00790=-118007,-112900,-122267,-13806,90840,35020
C00791=-118044,-112536,-122505,-13803,91159,34973
C00792=-118576,-105776,-120168,-13731,93052,34586
C00793=-118044,-112536,-122505,-13803,91159,34973
C00794=-125955,-111499,-122045,-12179,90192,32457
C00795=-127333,-111877,-122174,-11884,89885,32033
C00796=-124755,-111115,-121914,-12435,90480,32824
C00797=-119624,-116552,-128230,-13509,92325,34321
C00798=-117231,-121833,-124467,-22052,85463,28755
C00799=-122341,-114124,-118662,-20866,84531,27121
C00800=-123318,-113111,-117155,-20643,83910,26885
C00801=-123641,-113323,-116249,-20585,83205,26892
C00802=-123595,-112804,-116375,-20585,83540,26851
C00803=-123397,-106736,-114247,-20589,85286,26623
C00804=-123595,-112804,-116375,-20585,83540,26851
C00805=-116023,-114044,-115764,-22346,84523,29358
C00806=-117346,-116777,-115957,-22098,82979,29171
C00807=-118867,-116723,-116143,-21757,82713,28674
C00808=-116293,-116772,-115815,-22329,83179,29512
C00809=-117231,-121833,-124467,-22052,85463,28755
C00810=-154726,-134692,-133300,19029,79240,32627
C00811=-155157,-123239,-125350,19102,80279,32639
C00812=-155214,-122106,-123677,19140,79867,32554
C00813=-155216,-122330,-122794,19175,79245,32454
C00814=-155272,-122641,-123186,19186,79334,32449
C00815=-154565,-115790,-120970,18882,81218,32994
C00816=-155272,-122449,-123985,19155,79894,32538
C00817=-110972,-119209,-121408,-15853,79302,48266
C00818=-109086,-133769,-122042,-16854,72857,49812
C00819=-111848,-135958,-122676,-16103,71595,48979
C00820=-109086,-133769,-122042,-16854,72857,49812
C00821=-108592,-130707,-130810,-16554,79646,49045
C00822=-120610,-122471,-119242,-21572,81234,22537
C00823=-120610,-122484,-118172,-21604,80613,22649
C00824=-120610,-122391,-116483,-21658,79689,22817
C00825=-120610,-122419,-116833,-21647,79876,22783
C00826=-120610,-122423,-116832,-21647,79874,22783
C00827=-120610,-122419,-116833,-21647,79876,22783
C00828=-120610,-122416,-116761,-21649,79836,22790
C00829=-120610,-122436,-116768,-21650,79830,22791
C00830=-120610,-122416,-116761,-21649,79836,22790
C00831=-120611,-122370,-120508,-21535,82009,22397
C00832=-120500,-119354,-126515,-17332,87675,17755
C00833=-155157,-123239,-125350,19102,80279,32639
C00834=-155214,-122106,-123677,19140,79867,32554
C00835=-155216,-122330,-122794,19175,79245,32454
C00836=-155272,-122641,-123186,19186,79334,32449
C00837=-154565,-115790,-120970,18882,81218,32994
C00838=-155272,-122449,-123985,19155,79894,32538
C00839=-110972,-119209,-121408,-15853,79302,48266
C00840=-109086,-133769,-122042,-16854,72857,49812
C00841=-111848,-135958,-122676,-16103,71595,48979
C00842=-109086,-133769,-122042,-16854,72857,49812
C00843=-108592,-130707,-130810,-16554,79646,49045
C00844=-120611,-118687,-129075,-3134,90000,4412
C00845=-120611,-121772,-123926,-3138,85252,4531
C00846=-120611,-122092,-122744,-3141,84362,4553
C00847=-120611,-122362,-121169,-3146,83256,4581
C00848=-120611,-122286,-121724,-3144,83636,4571
C00849=-120611,-122290,-121724,-3144,83633,4571
C00850=-120611,-122286,-121724,-3144,83636,4571
C00851=-120611,-121006,-125813,-3134,86805,4492
C00852=-120621,-113915,-131911,-13153,116790,34478
C00853=-136832,-143297,-133894,-19017,104291,40845
C00854=-187686,-122249,-118318,-34521,102174,42234
C00855=-187703,-122088,-115580,-34298,100833,42653
C00856=-187707,-122010,-114917,-34250,100525,42749
C00857=-187713,-121734,-113169,-34135,99743,42991
C00858=-187707,-122010,-114917,-34250,100525,42749
C00859=-187770,-121697,-112491,-32279,113674,44764
C00860=-187767,-121692,-112491,-32279,113678,44765
C00861=-187770,-121697,-112491,-32279,113674,44764
C00862=-187667,-121438,-112064,-34928,84963,41689
C00863=-187673,-121448,-112068,-34927,84958,41688
C00864=-187667,-121438,-112064,-34928,84963,41689
C00865=-187641,-121360,-124129,-34919,91154,39753
C00866=-178673,-119471,-127738,-23493,103847,53429
C00867=-160878,-120510,-126471,-37,121976,81968
C00868=-160881,-121699,-123664,-37,119637,81967
C00869=-160883,-121991,-122485,-37,118762,81967
C00870=-160886,-122244,-120905,-37,117660,81966
C00871=-160884,-122111,-121864,-37,118318,81967
C00872=-160882,-122100,-121862,-36,118322,81968
C00873=-160884,-122111,-121864,-37,118318,81967
C00874=-160879,-120821,-125908,-37,121469,81968
C00875=-160879,-120821,-131564,-37,121469,81968
C00876=-157394,-128671,-131753,738,117538,83283
C00877=-158801,-138021,-132727,409,113343,82737
C00878=-158801,-138035,-132347,409,113101,82737
C00879=-158801,-138034,-131509,408,112586,82736
C00880=-158801,-138039,-131833,408,112783,82736
C00881=-160693,-149427,-134985,6,108877,82039
C00882=-160612,-153549,-136083,24,107435,82069
C00883=-159125,-144348,-133603,336,110634,82611
C00884=-199963,-104116,-119881,11013,127404,83152
C00885=-204692,-116225,-118816,8637,121169,80600
C00886=-203581,-121519,-120530,8810,119404,80895
C00887=-204849,-113790,-122122,8953,124435,80816
C00888=-166129,-114439,-129167,13521,133132,-54375
C00889=-82387,-124374,-130385,21792,102809,-55833
C00890=-37550,-124758,-124791,27166,84975,-54517
C00891=-35933,-124831,-122904,26864,83389,-54284
C00892=-35589,-124875,-121597,26827,82538,-54351
C00893=-35584,-124889,-121174,26839,82296,-54405
C00894=-35764,-126387,-121953,26892,82093,-54519
C00895=-31633,-125451,-121673,25972,81076,-53208
C00896=-35764,-126387,-121953,26892,82093,-54519
C00897=-46981,-157328,-126723,35790,81436,-33730
C00898=-42905,-153934,-122174,35701,78867,-32870
C00899=-42758,-143813,-119569,35389,81762,-31868
C00900=-42905,-153934,-122174,35701,78867,-32870
C00901=-53188,-117519,-120731,36414,97747,-30962
C00902=-95179,-109851,-129540,3422,106316,17944
C00903=-143691,-100776,-119079,-26047,122130,73021
C00904=-146029,-112499,-120098,-24937,116556,73463
C00905=-147204,-116618,-119576,-24569,113992,73590
C00906=-147487,-116577,-118677,-24502,113425,73607
C00907=-146967,-116625,-120319,-24630,114475,73574
C00908=-147345,-121113,-121824,-24401,113105,73737
C00909=-146899,-128254,-123879,-23878,111030,74376
C00910=-147345,-121113,-121824,-24401,113105,73737
C00911=-118081,-135478,-120686,-30293,109901,65237
C00912=-118366,-136707,-118609,-29972,108136,65614
C00913=-120887,-140213,-119894,-30302,106351,65070
C00914=-118366,-136707,-118609,-29972,108136,65614
C00915=-117820,-130449,-123242,-31209,113594,64262
C00916=-93926,-103398,-125362,-18301,106221,39936
C00917=-72688,-110808,-124077,-7134,85250,24096
C00918=-75848,-101444,-116923,-6191,85411,23073
C00919=-76170,-100985,-115528,-6097,84767,23002
C00920=-76167,-101481,-114835,-6104,84090,23035
C00921=-78739,-96930,-113773,-5320,85595,22140
C00922=-79843,-95445,-113201,-4985,85938,21775
C00923=-77748,-98228,-114268,-5620,85298,22470
C00924=-140085,-104632,-109249,40944,98797,-6712
C00925=-140263,-103640,-106572,40817,98007,-7102
C00926=-137942,-102173,-106029,40697,97269,-6378
C00927=-140263,-103640,-106572,40817,98007,-7102
C00928=-135988,-101428,-112112,41019,99549,-4631
C00929=-141957,-83285,-117139,12315,91699,6710
C00930=-161957,-129781,-122866,-20018,67926,12328
C00931=-166016,-109699,-113650,-17211,72980,10098
C00932=-166795,-105246,-111748,-16434,74862,9605
C00933=-165677,-113012,-111900,-18316,68836,10778
C00934=-162725,-116093,-113629,-19548,69016,11850
C00935=-162651,-107484,-110669,-19284,71494,11460
C00936=-162725,-116093,-113629,-19548,69016,11850
C00937=-155151,-112727,-112486,-22270,71877,14160
C00938=-155120,-113819,-110277,-22518,70103,14518
C00939=-159000,-114269,-110433,-21107,68960,13264
C00940=-155120,-113819,-110277,-22518,70103,14518
C00941=-155137,-138999,-124748,-23105,66364,15269
C00942=-81055,-115973,-127517,23586,109336,-64560
C00943=-76492,-127739,-126040,22738,101683,-64421
C00944=-76072,-128597,-125529,22671,100870,-64425
C00945=-76065,-128640,-125326,22657,100732,-64448
C00946=-76072,-128576,-125785,22685,101025,-64394
C00947=-82641,-146978,-130130,22016,96499,-67668
C00948=-81130,-155003,-132256,21951,93476,-67670
C00949=-82641,-146978,-130130,22016,96499,-67668
C00950=-84000,-144678,-127518,21929,96467,-68175
C00951=-84000,-143983,-126065,21900,95967,-68269
C00952=-83327,-146231,-127404,21916,95478,-68108
C00953=-88356,-135439,-132684,22407,104994,-68175
C00954=-104080,-128245,-132212,-31995,84146,-22143
C00955=-106783,-105266,-117364,-31197,85468,-23533
C00956=-107129,-103609,-115494,-31111,85090,-23558
C00957=-107127,-104217,-114421,-31144,84251,-23329
C00958=-107044,-104571,-114816,-31164,84333,-23320
C00959=-107880,-99055,-112779,-30885,85404,-23924
C00960=-107044,-104571,-114816,-31164,84333,-23320
C00961=-105114,-115284,-123193,-31689,84721,-22698
C00962=-105208,-113465,-123990,-31624,85910,-23065
C00963=-106823,-104635,-117017,-31184,85549,-23570
C00964=-107122,-103295,-115264,-31113,85109,-23561
C00965=-107121,-103855,-114286,-31142,84342,-23351
C00966=-107087,-104437,-114776,-31151,84356,-23343
C00967=-107921,-98925,-112738,-30873,85426,-23945
C00968=-107087,-104437,-114776,-31151,84356,-23343
C00969=-105701,-116384,-125830,-31502,85418,-23114
C00970=-63541,-120749,-127234,-38861,101172,-11499
C00971=-62914,-102725,-115578,-39257,103083,-11954
C00972=-62914,-103574,-114098,-39030,102025,-11552
C00973=-62914,-103512,-114221,-39048,102111,-11585
C00974=-65395,-98857,-112499,-39034,102095,-12627
C00975=-63190,-103387,-116908,-39318,103341,-12168
C00976=-105701,-116384,-125830,-31502,85418,-23114
C00977=-79137,-116524,-127291,-7118,77084,38210
C00978=-66518,-158449,-133200,-8588,59166,50817
C00979=-70166,-147728,-127011,-6864,60501,49298
C00980=-71549,-143558,-123868,-6244,60595,48757
C00981=-71544,-142942,-122687,-6271,60188,48782
C00982=-71412,-140542,-122600,-6259,61371,48766
C00983=-74130,-137647,-121783,-5023,62161,47690
C00984=-71412,-140542,-122600,-6259,61371,48766
C00985=-59221,-85077,-106862,-19044,97138,55247
C00986=-59772,-90133,-108950,-18878,95774,55276
C00987=-59221,-85077,-106862,-19044,97138,55247
C00988=-65406,-128676,-128270,-8670,80773,42177
C00989=-57064,-112054,-129147,-2862,108793,29097
C00990=-70948,-123089,-127271,10962,111372,-380
C00991=-67644,-116564,-123033,11394,111660,848
C00992=-67644,-116773,-122597,11361,111292,811
C00993=-67644,-116291,-123546,11437,112109,893
C00994=-70770,-123262,-125779,10903,110357,-412
C00995=-70770,-123588,-124717,10837,109552,-488
C00996=-69306,-120453,-123728,11077,110342,115
C00997=-70770,-123283,-125719,10898,110311,-416
C00998=-70770,-119886,-130778,11344,115083,53
C00999=-68413,-122856,-123349,22437,117236,58
C01000=-67404,-122631,-120786,22344,115611,123
C01001=-67401,-122683,-120099,22253,115193,37
C01002=-67283,-122594,-120333,22317,115338,115
C01003=-65261,-118175,-118917,23034,116088,1096
C01004=-67283,-122594,-120333,22317,115338,115
C01005=-70820,-123560,-126018,22187,119059,-540
C01006=-59587,-128850,-129971,-18356,103459,48793
C01007=-60648,-112549,-116046,-37363,97913,74718
C01008=-66648,-121539,-115269,-36526,91263,74498
C01009=-69624,-125916,-115212,-36242,88151,74300
C01010=-69624,-125773,-114639,-36242,87924,74374
C01011=-69624,-125814,-114800,-36242,87987,74354
C01012=-70738,-127677,-115368,-36152,87024,74211
C01013=-69624,-125814,-114800,-36242,87987,74354
C01014=-61556,-115340,-115782,-37136,96245,74919
C01015=-93863,-107857,-129738,-18786,98098,27923
C01016=-113340,-105978,-120535,-17383,92037,15860
C01017=-116256,-99504,-115214,-16745,91512,14962
C01018=-117355,-97038,-113094,-16498,91266,14630
C01019=-124053,-106600,-116618,-14934,87391,12894
C01020=-123019,-109757,-118902,-15179,87365,13243
C01021=-120254,-118381,-124729,-15823,87055,14212
C01022=-121076,-118719,-112405,-41381,81563,9211
C01023=-125328,-110839,-107644,-40465,80446,7775
C01024=-126920,-107772,-105722,-40091,80023,7243
C01025=-122279,-105715,-102241,-45382,81605,7865
C01026=-118123,-103314,-98388,-50429,83325,8212
C01027=-115452,-99808,-95169,-50805,84680,8860
C01028=-113598,-101964,-96694,-51043,85596,9323
C01029=-108732,-107177,-100380,-51565,88044,10518
C01030=-131658,-113091,-133069,-11905,90618,-13395
C01031=-155934,-143784,-122811,23124,58745,-32427
C01032=-151507,-132468,-117411,20635,59886,-30339
C01033=-149876,-128251,-115276,19729,60288,-29596
C01034=-151213,-128323,-114307,20456,60014,-30191
C01035=-146890,-120795,-114089,13688,65901,-25886
C01036=-142734,-111238,-112703,7950,73001,-22079
C01037=-143750,-114926,-115045,8343,72653,-22456
C01038=-146492,-125018,-121022,9420,71459,-23506
C01039=-146459,-122334,-129315,9145,77857,-23007
C01040=-118526,-115013,-133262,8809,105739,-46794
C01041=-93674,-118800,-129721,8134,120991,-68616
C01042=-93669,-120967,-127104,7892,118292,-68817
C01043=-94465,-127736,-127937,7493,115415,-69310
C01044=-101667,-152205,-134731,5550,107657,-72408
C01045=-93660,-121042,-127131,7893,118270,-68815
C01046=-93665,-118880,-129750,8134,120967,-68614
C01047=-98446,-113408,-116165,41475,93741,-73013
C01048=-95217,-118830,-115137,40946,89638,-73223
C01049=-92806,-121560,-115150,40665,87459,-73017
C01050=-95954,-130241,-115077,41081,85472,-75169
C01051=-96936,-125131,-114749,41104,87782,-74702
C01052=-101504,-121000,-116278,41571,92256,-74948
C01053=-100864,-122088,-112493,43204,76282,-71688
C01054=-96953,-122826,-110054,42689,72984,-71279
C01055=-94247,-124338,-109802,42269,70974,-70864
C01056=-94193,-123974,-108080,42453,70297,-71131
C01057=-95642,-121622,-108630,42447,72155,-71017
C01058=-100864,-121830,-111367,43291,75868,-71867
C01059=-131033,-115476,-133015,2815,101744,-74384
C01060=-151471,-119125,-123137,-34971,103386,-73225
C01061=-162012,-101235,-114016,-37763,108592,-75954
C01062=-165297,-105997,-114400,-37202,105452,-76208
C01063=-161279,-107047,-112450,-36906,105725,-74600
C01064=-157962,-101866,-111865,-37402,108959,-74341
C01065=-155898,-93647,-112180,-38609,113341,-75115
C01066=-93674,-112333,-133466,8753,126560,-68151
C01067=-93674,-118800,-129721,8134,120991,-68616
C01068=-93669,-120967,-127104,7892,118292,-68817
C01069=-93667,-121558,-126026,7814,117333,-68886
C01070=-93663,-121536,-126144,7822,117416,-68879
C01071=-93639,-121762,-126135,7818,117296,-68878
C01072=-93680,-121434,-126040,7817,117406,-68885
C01073=-93660,-121042,-127131,7893,118270,-68815
C01074=-93665,-118880,-129750,8134,120967,-68614
C01075=-98446,-113408,-116165,41475,93741,-73013
C01076=-93996,-117843,-114815,40802,89312,-72817
C01077=-91343,-117266,-113836,40455,87860,-72224
C01078=-92137,-119395,-114109,40564,87510,-72703
C01079=-95072,-126184,-113786,40951,86041,-74561
C01080=-95071,-125918,-112907,40977,85731,-74679
C01081=-96936,-125131,-114749,41104,87782,-74702
C01082=-101504,-121000,-116278,41571,92256,-74948
C01083=-100864,-122088,-112493,43204,76282,-71688
C01084=-95643,-121963,-109784,42340,72556,-70846
C01085=-93677,-120964,-108398,41948,71358,-70433
C01086=-93599,-120925,-107098,42100,70733,-70661
C01087=-95642,-121622,-108630,42447,72155,-71017
C01088=-100864,-121830,-111367,43291,75868,-71867
C01089=-131033,-115476,-133015,2815,101744,-74384
C01090=-151471,-119125,-123137,-34971,103386,-73225
C01091=-162012,-101235,-114016,-37763,108592,-75954
C01092=-163593,-104354,-113811,-37340,106547,-75879
C01093=-162938,-104376,-113793,-37349,106803,-75692
C01094=-158829,-104862,-111593,-37019,107224,-74083
C01095=-157962,-101866,-111865,-37402,108959,-74341
C01096=-155898,-93647,-112180,-38609,113341,-75115
C01097=-179206,-139250,-107986,-62075,77828,-66561
C01098=-185232,-138953,-105140,-62379,73225,-66913
C01099=-187696,-139015,-104542,-62453,71468,-67163
C01100=-187702,-137665,-102648,-62587,71237,-66963
C01101=-185238,-138055,-103864,-62461,73065,-66778
C01102=-179211,-138396,-106727,-62132,77661,-66424
C01103=-179188,-148562,-121526,-61524,79591,-68010
C01104=-184417,-115822,-131978,-19629,107310,7500
C01105=-190427,-134899,-136820,8574,116374,78562
C01106=-188066,-120573,-128029,9218,118052,79593
C01107=-191610,-147357,-136376,6897,103791,75181
C01108=-187795,-119828,-126345,9210,117376,79639
C01109=-187841,-121664,-124728,-2971,114560,78170
C01110=-187942,-121398,-126015,-3016,115485,78109
C01111=-187937,-119495,-128851,-3098,118205,78035
C01112=-176042,-128909,-129640,-7380,110692,58022
C01113=-187833,-113452,-115854,-34994,105139,41767
C01114=-187847,-113781,-113588,-34722,103839,42187
C01115=-187853,-113844,-112659,-34623,103335,42348
C01116=-187856,-113866,-111596,-34519,102780,42525
C01117=-187851,-113844,-112538,-34611,103274,42368
C01118=-187836,-113627,-114840,-34866,104547,41960
C01119=-186756,-108501,-120882,-36201,110201,40487
C01120=-150585,-129060,-123753,-46684,114085,-39870
C01121=-134046,-137019,-115206,-49635,112096,-74674
C01122=-134033,-140586,-110307,-48065,108843,-72866
C01123=-134037,-138671,-107458,-47843,108316,-72589
C01124=-133950,-137111,-106105,-47812,108341,-72556
C01125=-133930,-150358,-126108,1173,113974,-57522
C01126=-134040,-150029,-126001,1133,114079,-57562
C01127=-134505,-148512,-125722,2741,114238,-57140
C01128=-137673,-151162,-132623,1623,117206,-58299
C01129=-106012,-107394,-121753,14018,130776,-44816
C01130=-106669,-102485,-112824,13121,127987,-45519
C01131=-97512,-96218,-110425,14566,129183,-82759
C01132=-98864,-105619,-112306,13303,125832,-83842
C01133=-106150,-109468,-113796,12766,125107,-45727
C01134=-105474,-116823,-114648,29161,97726,-33837
C01135=-134074,-146851,-118858,40485,90771,-46834
C01136=-141855,-151854,-132376,33568,89282,-32323
C01137=-173958,-148748,-133240,11874,65312,15203
C01138=-187653,-128002,-123664,-7056,57779,46476
C01139=-188071,-112180,-99768,1790,31671,46486
C01140=-188092,-111455,-97340,1875,30550,46442
C01141=-187851,-111485,-96835,1581,30220,46589
C01142=-187792,-110201,-93997,1555,29133,46605
C01143=-187737,-110060,-93474,1490,28882,46636
C01144=-187785,-109075,-90961,1604,27844,46576
C01145=-188106,-109627,-92159,2030,28303,46362
C01146=-188086,-110531,-94662,1935,29378,46411
C01147=-188086,-114129,-114927,1479,39995,46659
C01148=-201470,-41376,-102585,19941,97743,-57993
C01149=-197439,-2624,-49840,39121,107911,-51008
C01150=-168348,92819,48556,27514,116832,-48709
C01151=-170146,82769,36005,28011,119675,-48673
C01152=-172466,59662,8523,30747,114377,-38085
C01153=-173361,44293,-8668,31536,116980,-37634
C01154=-173326,42548,-10417,31798,119739,-39927
C01155=-173293,31446,-22173,31559,124382,-42741
C01156=-170045,43132,-9775,28753,130915,-51393
C01157=-186843,33187,-28183,45340,118495,-56566
C01158=-187270,22965,-40018,42118,113549,-44205
C01159=-164927,12374,-50848,37497,97302,26684
C01160=-160848,-52651,-98971,6904,73590,44156
C01161=-187933,-111679,-98706,-278,30585,46526
C01162=-187953,-110958,-96368,-260,29517,46517
C01163=-188171,-110591,-95666,34,29272,46369
C01164=-188111,-109885,-93130,-50,28074,46412
C01165=-188090,-109778,-92606,-82,27808,46427
C01166=-188055,-108797,-90194,-133,26826,46455
C01167=-187968,-109087,-91174,-258,27282,46516
C01168=-187948,-109974,-93584,-278,28309,46526
C01169=-190713,-138118,-122139,3147,45685,54861
C01170=-188097,-104568,-127563,3199,90457,72619
C01171=-188112,-108983,-124849,3203,86524,72515
C01172=-196049,-130715,-128058,11352,73875,69900
C01173=-196049,-130372,-129815,11289,75109,70015
C01174=-199069,-128516,-127529,12349,75098,68966
C01175=-193131,-119078,-125609,7963,80164,71095
C01176=-187364,-124777,-127140,2732,76642,72458
C01177=-191510,-130298,-128202,6704,73471,71168
C01178=-188153,-109076,-124888,3215,86502,72501
C01179=-188138,-104664,-127604,3212,90434,72606
C01180=-187898,-111965,-120493,-16766,69565,69566
C01181=-187918,-113285,-117348,-17044,67055,69927
C01182=-188433,-114855,-116277,-16981,65546,69965
C01183=-188279,-112660,-115510,-16972,66207,69918
C01184=-188347,-112560,-115415,-16943,66188,69897
C01185=-188064,-112094,-115237,-17061,66369,69976
C01186=-187944,-113344,-117352,-17035,67023,69922
C01187=-187924,-112030,-120500,-16757,69531,69561
C01188=-180038,-109975,-126789,-2440,82512,-7441
C01189=-174468,-102021,-118148,-1871,82653,-17547
C01190=-174479,-103807,-115834,-1877,80312,-17516
C01191=-175021,-104384,-114967,-1695,79470,-17680
C01192=-174783,-104250,-115053,-1777,79597,-17606
C01193=-174170,-106690,-109656,-11758,69864,-18312
C01194=-172833,-107431,-109671,-12341,69693,-17819
C01195=-174390,-105691,-110273,-11607,70709,-18474
C01196=-174377,-104937,-112785,-11492,72607,-18653
C01197=-190845,-100837,-124447,13698,93294,-33124
C01198=-206306,-116062,-120388,37359,88631,-50073
C01199=-215039,-120395,-106715,50971,83253,-62053
C01200=-215038,-119729,-104733,51036,82687,-62365
C01201=-215037,-119445,-103934,51064,82464,-62488
C01202=-215047,-118488,-101366,51160,81769,-62880
C01203=-215047,-118800,-102176,51129,81987,-62759
C01204=-215049,-119543,-104187,51057,82539,-62453
C01205=-215012,-122438,-115563,50746,86080,-60488
C01206=-160845,-113405,-113287,47121,77099,31472
C01207=-160851,-113463,-110064,47446,75709,30781
C01208=-161105,-114307,-109195,47677,75177,30385
C01209=-161122,-114371,-109216,47688,75170,30377
C01210=-115363,-119356,-110747,30444,52974,43110
C01211=-116247,-123536,-113883,31027,53106,42730
C01212=-160782,-112987,-114684,46949,77813,31850
C01213=-161690,-87231,-108001,36248,90547,80444
C01214=-156405,-91013,-102041,34922,83859,80351
C01215=-152529,-73393,-94338,33696,85968,82496
C01216=-158330,-83683,-104653,35339,89043,81248
C01217=-160758,-112853,-114863,36163,82877,78288
C01218=-160760,-113152,-111426,36317,81029,77674
C01219=-159491,-108015,-113138,31549,97627,78488
C01220=-160866,-112928,-114836,31527,96856,77736
C01221=-163914,-124233,-119408,29285,98886,76856
C01222=-164622,-129006,-121133,28240,99357,76613
C01223=-160757,-112482,-116558,30024,102576,77779
C01224=-160755,-111254,-119690,30396,104801,78387
C01225=-139139,-104942,-132434,5076,105021,81413
C01226=-120610,-140892,-128239,-26796,83300,73925
C01227=-124485,-139346,-124335,-26282,80622,73071
C01228=-128794,-174695,-130569,-28116,58521,76693
C01229=-123854,-173705,-127920,-33486,56775,79744
C01230=-127596,-155142,-123084,-28725,56836,77726
C01231=-128095,-155529,-122172,-29132,53686,78388
C01232=-128860,-155984,-126780,-25446,58633,74277
C01233=-138109,-135032,-133743,-8289,74304,51513
C01234=-203654,-125968,-124215,37381,73551,-30645
C01235=-201127,-103516,-110680,20461,62884,-59060
C01236=-201138,-104157,-107983,20829,61019,-59420
C01237=-201193,-104400,-106652,21043,60147,-59612
C01238=-201232,-104446,-106694,21063,60161,-59627
C01239=-200873,-105228,-106882,20926,59802,-59552
C01240=-201116,-104130,-107973,20816,61021,-59411
C01241=-201105,-103488,-110669,20449,62886,-59051
C01242=-198523,-119273,-121454,24683,77158,-64296
C01243=-174403,-100049,-121231,21877,99309,-62114
C01244=-174406,-102879,-118773,21681,96545,-62622
C01245=-172958,-103152,-117900,21399,95556,-62302
C01246=-174224,-104881,-115910,21520,93897,-63036
C01247=-174418,-104205,-117181,21599,94999,-62906
C01248=-174415,-101880,-119808,21752,97619,-62429
C01249=-185776,-93152,-118465,-1785,83350,-67432
C01250=-169060,-142396,-123848,-37084,49654,-60484
C01251=-174230,-113472,-108308,-34615,49911,-64397
C01252=-174247,-112967,-104740,-35556,48304,-63744
C01253=-174471,-112928,-103062,-35946,47380,-63468
C01254=-174489,-112275,-102294,-36008,47261,-63425
C01255=-174590,-112153,-101603,-36140,46922,-63333
C01256=-174396,-113097,-100663,-36857,46141,-62871
C01257=-174330,-114043,-100633,-37190,45762,-62656
C01258=-174129,-122060,-98220,-45554,37107,-60115
C01259=-174246,-112406,-102200,-36228,47262,-63291
C01260=-174229,-113129,-105847,-35265,48804,-63944
C01261=-182962,-136134,-123657,-29797,44727,-67038
C01262=-203654,-125968,-124215,37381,73551,-30645
C01263=-201127,-103516,-110680,20461,62884,-59060
C01264=-201138,-104157,-107983,20829,61019,-59420
C01265=-201193,-104400,-106652,21043,60147,-59612
C01266=-201232,-104446,-106694,21063,60161,-59627
C01267=-200873,-105228,-106882,20926,59802,-59552
C01268=-201116,-104130,-107973,20816,61021,-59411
C01269=-201105,-103488,-110669,20449,62886,-59051
C01270=-198523,-119273,-121454,24683,77158,-64296
C01271=-174403,-100049,-121231,21877,99309,-62114
C01272=-174406,-102879,-118773,21681,96545,-62622
C01273=-172958,-103152,-117900,21399,95556,-62302
C01274=-174224,-104881,-115910,21520,93897,-63036
C01275=-174418,-104205,-117181,21599,94999,-62906
C01276=-174415,-101880,-119808,21752,97619,-62429
C01277=-185776,-93152,-118465,-1785,83350,-67432
C01278=-169060,-142396,-123848,-37084,49654,-60484
C01279=-174230,-113472,-108308,-34615,49911,-64397
C01280=-174247,-112967,-104740,-35556,48304,-63744
C01281=-174471,-112928,-103062,-35946,47380,-63468
C01282=-174489,-112275,-102294,-36008,47261,-63425
C01283=-174590,-112153,-101603,-36140,46922,-63333
C01284=-174396,-113097,-100663,-36857,46141,-62871
C01285=-174330,-114043,-100633,-37190,45762,-62656
C01286=-174129,-122060,-98220,-45554,37107,-60115
C01287=-174246,-112406,-102200,-36228,47262,-63291
C01288=-175798,-117006,-109100,-34199,48210,-64559
C01289=-178617,-124532,-114828,-32467,46840,-65534
C01290=-210827,-121899,-127370,-35396,86436,-76908
C01291=-214505,-124636,-123608,-35577,86411,-76994
C01292=-214521,-124823,-120077,-35640,84542,-76397
C01293=-209595,-138372,-118962,-40572,76618,-76704
C01294=-215572,-134536,-117924,-37557,71164,-81051
C01295=-214545,-124844,-120083,-35636,84527,-76402
C01296=-214528,-124659,-123615,-35573,86395,-76999
C01297=-214596,-124890,-121786,-39550,96156,-78039
C01298=-214607,-124784,-118461,-39383,94595,-77461
C01299=-215336,-122839,-115954,-39308,93846,-77495
C01300=-215216,-123286,-113688,-39218,92622,-76995
C01301=-214785,-119888,-114308,-39371,94481,-77497
C01302=-214619,-124823,-118761,-39395,94718,-77513
C01303=-214540,-124430,-116246,-48349,86426,-68042
C01304=-214499,-123956,-126099,-48385,90728,-70182
C01305=-158797,-145907,-128305,-56145,74291,-56792
C01306=-118138,-117595,-113507,-59219,64127,-52420
C01307=-134091,-119062,-102284,-58108,50235,-52331
C01308=-134095,-117716,-98836,-59129,49460,-51612
C01309=-134657,-117185,-97454,-59366,48806,-51448
C01310=-134083,-121591,-110246,-11584,43366,-62365
C01311=-133895,-121523,-110170,-11744,43379,-62274
C01312=-133843,-121378,-109751,-11603,42967,-62923
C01313=-134088,-120272,-105685,-8075,39028,-71413
C01314=-134097,-120880,-107281,-7954,39689,-71484
C01315=-133538,-122024,-122159,-7272,48238,-71950
C01316=-134045,-120979,-109361,-39707,45136,-55893
C01317=-134048,-117179,-98466,-43015,41514,-53843
C01318=-133905,-117568,-98535,-40781,40764,-54269
C01319=-134181,-118830,-102497,-12918,37668,-61575
C01320=-134198,-119226,-102647,-12934,37556,-61565
C01321=-167359,-106948,-94294,44068,50330,-74802
C01322=-162364,-123197,-107171,35832,43944,-75497
C01323=-134045,-120979,-109361,-39707,45136,-55893
C01324=-132003,-121638,-109572,-41117,45917,-55073
C01325=-131002,-106489,-98392,-41164,47077,-55091
C01326=-131123,-103588,-88252,-50265,40796,-51296
C01327=-163242,-98975,-95762,18008,45953,-74760
C01328=-153405,-104865,-97946,10266,42608,-70493
C01329=-134148,-119761,-102793,-13034,37388,-61506
C01330=-126986,-126229,-93303,56145,28917,-85918
C01331=-131099,-132353,-104040,54087,33374,-85008
C01332=-133651,-114033,-99266,51853,45977,-77066
C01333=-134816,-132236,-131789,-6177,48808,-72548
C01334=-152519,-98596,-126841,-17039,86437,-59409
C01335=-167034,-82548,-116958,-26153,108191,-47353
C01336=-167227,-85698,-113927,-25595,104988,-46679
C01337=-155614,-79416,-105751,-37322,108167,-45505
C01338=-159401,-74916,-103736,-37095,107545,-46814
C01339=-167994,-62773,-97902,-36298,106416,-49798
C01340=-170767,-58288,-95591,-35952,106111,-50754
C01341=-180979,-58723,-101497,-23976,107062,-51805
C01342=-180909,-54943,-104050,-24554,110296,-52487
C01343=-168157,-75412,-102271,-33648,91006,-21456
C01344=-174012,-67106,-91297,-33471,82630,-14810
C01345=-175466,-61382,-85667,-32996,81659,-15067
C01346=-176013,-59150,-83405,-32819,81253,-15153
C01347=-202608,-62025,-89962,4221,78254,-36710
C01348=-159972,-87195,-101610,-14286,75081,-22762
C01349=-154310,-93015,-102157,-19304,70769,-24486
C01350=-154362,-96202,-104591,-19297,70625,-24481
C01351=-154503,-104813,-110762,-19306,69999,-24428
C01352=-155575,-73729,-96860,-32555,86012,-14938
C01353=-157088,-68154,-91284,-32096,84992,-15206
C01354=-157731,-66276,-89193,-31903,84490,-15302
C01355=-176839,-77218,-97385,-7105,75561,-28432
C01356=-165473,-80321,-98709,-11948,76053,-24715
C01357=-199796,-81518,-91231,35244,71315,-57262
C01358=-201423,-82172,-92479,35779,72324,-57601
C01359=-205660,-83542,-95477,37134,74990,-58446
C01360=-150225,-90058,-124320,-20069,81923,-14603
C01361=-88917,-116100,-126028,-29630,66347,39612
C01362=-48102,-114880,-112674,-35477,56596,75725
C01363=-53396,-105773,-101201,-33500,52497,74682
C01364=-53385,-105323,-98106,-34230,51099,75219
C01365=-48465,-101460,-95464,-40425,56724,79171
C01366=-72122,-108844,-98440,461,39847,55622
C01367=-53363,-105522,-99057,-19217,46878,60217
C01368=-53371,-105892,-101942,-18746,48378,59901
C01369=-53322,-113038,-104699,812,43724,42660
C01370=-53318,-112442,-102021,830,42382,42650
C01371=-53317,-112163,-100935,837,41857,42645
C01372=-53253,-112229,-97736,1547,37461,42516
C01373=-53300,-111445,-98358,1568,38246,42506
C01374=-51520,-115460,-104005,-179,39644,43460
C01375=-55761,-139961,-122674,-27476,66843,55729
C01376=-53542,-121644,-113892,-40363,83761,61539
C01377=-53523,-121175,-111327,-40444,82737,61941
C01378=-53533,-120846,-110023,-41635,87424,59647
C01379=-53533,-120798,-109834,-41636,87355,59676
C01380=-53529,-120315,-108043,-41648,86710,59935
C01381=-53536,-120580,-109029,-41640,87063,59791
C01382=-53556,-121151,-111460,-41628,87965,59422
C01383=-52633,-122748,-126719,-40391,89833,59612
C01384=-140119,-108661,-130674,-21165,82789,-25459
C01385=-161125,-123349,-120158,-18581,66270,-46079
C01386=-131164,-149034,-123827,-31550,65486,-33807
C01387=-135268,-120375,-120219,-10307,79463,-36863
C01388=-120772,-128591,-116633,-33078,74633,-32200
C01389=-135999,-133464,-117919,-29207,67526,-36426
C01390=-160269,-123865,-115188,-19445,63316,-45243
C01391=-162856,-121662,-114495,-18189,63396,-46272
C01392=-161212,-123488,-116538,-18871,64068,-45743
C01393=-161202,-123677,-120265,-18562,66156,-46089
C01394=-167124,-146469,-125858,32695,63076,-70922
C01395=-161220,-122264,-110536,44525,64077,-74742
C01396=-161219,-121375,-107584,44985,63095,-75224
C01397=-164956,-113855,-102560,48427,66781,-75111
C01398=-161213,-120936,-106323,43985,60856,-74418
C01399=-161480,-119492,-104017,44742,56174,-74995
C01400=-161477,-119788,-101535,47560,52624,-77093
C01401=-161197,-119682,-102993,46927,53134,-76618
C01402=-161197,-120736,-105876,46275,53998,-76117
C01403=-161177,-121556,-108554,35078,57327,-43050
C01404=-161177,-120932,-106617,35398,56609,-43319
C01405=-152937,-127654,-109782,25136,48983,-42100
C01406=-161176,-119640,-103030,36318,54707,-44163
C01407=-161179,-121241,-107541,34339,64662,-45277
C01408=-161179,-121533,-108462,34233,65010,-45160
C01409=-161180,-122193,-110741,33972,65899,-44866
C01410=-159909,-111206,-128347,-10927,59798,-43136
C01411=-174276,-119239,-128019,9099,73009,32604
C01412=-174287,-122281,-118814,9519,65873,32039
C01413=-174304,-122135,-115653,9666,64029,31878
C01414=-174310,-121974,-114355,9727,63324,31815
C01415=-174277,-122172,-120616,-9764,82080,37769
C01416=-174277,-122177,-120568,-9764,82048,37772
C01417=-174317,-121775,-113110,-33515,107538,43031
C01418=-174312,-121937,-114098,-33622,107981,42892
C01419=-174299,-122214,-116525,-33911,109120,42531
C01420=-174287,-119835,-127268,-36019,115609,40290
C01421=-174287,-120021,-127206,9145,72119,32532
C01422=-174287,-120021,-127206,9145,72119,32532
C01423=-173736,-117333,-114872,9262,65925,32245
C01424=-174960,-111711,-111152,9771,66659,31859
C01425=-176831,-126585,-121826,-8311,79476,36809
C01426=-157010,-133467,-117360,-32643,99223,56368
C01427=-157552,-135759,-118018,-32604,98358,56401
C01428=-154345,-130153,-124672,-33336,105500,55567
C01429=-146682,-141770,-131473,-27794,101884,56245
C01430=-146682,-141770,-131473,-27794,101884,56245
C01431=-146682,-141770,-131473,15257,98468,53705
C01432=-102938,-141770,-131473,49664,98468,53705
C01433=-102938,-145417,-131473,49512,65454,53705
C01434=-103656,-129714,-109721,51674,62395,51470
C01435=-102995,-138917,-102303,63406,51064,43511
C01436=-104839,-135559,-111699,50177,75701,60454
C01437=-99828,-171084,-120161,53403,64595,56658
C01438=-110163,-126067,-103455,56717,91063,66073
C01439=-116435,-131456,-112749,56730,96510,65994
C01440=-116383,-133294,-113279,56655,96128,65766
C01441=-84454,-125099,-129012,35107,90636,33075
C01442=-15972,-110889,-128286,-10965,59905,-43045
C01443=-15972,-110889,-128286,-10965,59905,-43045
C01444=-53465,-86935,-89811,-40465,79071,68727
C01445=-108812,15435,-43443,-8262,104585,64007
C01446=-120685,104729,62045,12414,91835,74489
C01447=-120504,102152,62779,12366,90072,74374
C01448=-120431,101212,63194,12350,89339,74325
C01449=-120431,101002,64582,12347,88398,74232
C01450=-120431,101212,63194,12350,89339,74325
C01451=-121076,107244,72775,12456,86702,73844
C01452=-120665,102968,67176,12385,87860,74099
C01453=-121076,107271,71616,12453,87413,73914
C01454=-119318,105160,68851,12167,87755,74544
C01455=-119320,105991,71162,12170,86781,74448
C01456=-119694,104363,69033,12227,87301,74371
C01457=-119694,104435,67982,12226,87970,74437
C01458=-121323,110426,71256,12493,89251,74016
C01459=-131278,69881,50181,9127,63188,62805
C01460=-131485,74883,60411,9547,59533,62414
C01461=-131548,76399,63510,9674,58426,62296
C01462=-131548,76704,64506,9721,57977,62255
C01463=-131183,71204,57206,9397,59578,62541
C01464=-131183,71498,58283,9446,59073,62497
C01465=-131266,74091,61533,9552,58423,62408
C01466=-131382,69379,53589,9372,60872,62574
C01467=-130781,63634,40058,8705,66118,63219
C01468=-132526,40318,17232,-3897,63337,79864
C01469=-132770,43850,25861,-3900,59836,79894
C01470=-132775,45020,27808,-3921,59239,79913
C01471=-132775,45119,28557,-3937,58830,79928
C01472=-131974,40901,23457,-4303,59840,80201
C01473=-131974,40988,24219,-4322,59418,80218
C01474=-132343,43569,27070,-4148,58978,80090
C01475=-132425,41720,24361,-4076,59689,80031
C01476=-131916,36045,14544,-4216,62827,80109
C01477=-154350,3292,-38754,752,86522,75713
C01478=-181553,89062,52820,1715,95022,75090
C01479=-181735,85640,53357,1725,92938,75001
C01480=-181765,85113,53499,1727,92580,74986
C01481=-181767,85098,55139,1725,91564,74972
C01482=-181765,85113,53499,1727,92580,74986
C01483=-181351,93067,65191,1686,89465,75083
C01484=-181572,88775,59771,1706,90599,75024
C01485=-181351,93067,65191,1686,89465,75083
C01486=-181147,96755,64289,1671,91909,75184
C01487=-159394,22511,-602,-1012,64107,82504
C01488=-159231,25736,7387,-1125,60850,82595
C01489=-159102,29806,11901,-1198,60164,82651
C01490=-159102,29893,13040,-1208,59512,82655
C01491=-159102,29869,12753,-1208,59677,82655
C01492=-159322,25425,8401,-1088,60068,82565
C01493=-159448,23983,7363,-1023,59965,82516
C01494=-159276,26818,10107,-1116,59735,82583
C01495=-159294,26208,9511,-1106,59788,82576
C01496=-159294,26230,9792,-1106,59626,82576
C01497=-159101,23920,6361,-1196,60552,82648
C01498=-159295,23244,6238,-1098,60277,82577
C01499=-159295,23301,7050,-1101,59807,82580
C01500=-159299,25281,8955,-1100,59652,82580
C01501=-159295,23278,6733,-1101,59990,82580
C01502=-159427,17860,-3265,-1001,63356,82499
C01503=-180998,44453,11386,9428,69103,75000
C01504=-180806,46143,18147,9552,65832,74803
C01505=-180618,49143,21508,9515,65295,74827
C01506=-180618,49076,22901,9581,64417,74754
C01507=-180618,49087,22593,9566,64610,74771
C01508=-181106,45329,18547,9757,65218,74643
C01509=-181106,45312,18870,9772,65014,74625
C01510=-180958,47165,20854,9721,64729,74655
C01511=-180909,46562,20206,9690,64811,74680
C01512=-180909,46552,20476,9701,64642,74667
C01513=-180909,46563,20203,9689,64813,74682
C01514=-181219,43931,17395,9810,65220,74603
C01515=-181219,43906,17870,9834,64920,74577
C01516=-181012,45777,19861,9753,64635,74629
C01517=-181381,44679,17515,9863,65546,74571
C01518=-181427,38720,7071,9647,68865,74830
C01519=-152316,-9212,-39627,-4041,74028,47424
C01520=-97675,-116344,-75406,-30929,43249,-3453
C01521=-144147,-96317,-43020,16665,22045,18189
C01522=-130185,-5552,7433,-2044,36537,82607
C01523=-148170,9866,-4864,-2727,74191,81047
C01524=-160677,16615,-6140,-3325,93789,80088
C01525=-160892,14618,-3978,-3294,91428,80078
C01526=-160979,13901,-3035,-3283,90476,80074
C01527=-160979,13973,-1608,-3282,89636,80096
C01528=-160979,13952,-1963,-3282,89844,80091
C01529=-161075,20354,3961,-3273,89483,80067
C01530=-161075,20386,4410,-3273,89224,80073
C01531=-161133,18273,2432,-3268,89353,80049
C01532=-161218,18655,2789,-3260,89326,80020
C01533=-161218,18671,3009,-3260,89200,80024
C01534=-161218,18657,2809,-3260,89316,80021
C01535=-161242,21197,5196,-3258,89153,80017
C01536=-161242,21225,5559,-3258,88944,80022
C01537=-161222,19566,3996,-3259,89054,80025
C01538=-161093,20062,3160,-3271,89826,80048
C01539=-160610,22295,943,-3323,92353,80148
C01540=-159769,-26352,-42847,7626,75430,42908
C01541=-160661,-23608,-37245,8003,73495,42476
C01542=-161092,-17751,-31188,8180,72827,42281
C01543=-161092,-17734,-30227,8206,72247,42243
C01544=-161092,-17740,-30493,8199,72405,42254
C01545=-161118,-21273,-33081,8218,72187,42230
C01546=-161118,-21265,-32749,8226,71987,42217
C01547=-161116,-19976,-31814,8223,72071,42223
C01548=-161133,-20273,-32030,8231,72055,42216
C01549=-161133,-20265,-31761,8239,71896,42206
C01550=-161133,-20272,-31998,8233,72037,42215
C01551=-161051,-23031,-33989,8213,71838,42230
C01552=-161051,-23018,-33649,8222,71636,42217
C01553=-160924,-21492,-32553,8173,71734,42269
C01554=-161101,-22161,-33921,8213,72245,42241
C01555=-159612,-30937,-44211,7622,73912,42867
C01556=-144117,-44081,-61004,-17211,89666,8724
C01557=-145648,-40124,-55468,-16926,88039,8426
C01558=-146237,-38515,-53215,-16819,87384,8313
C01559=-146244,-38444,-53170,-16818,87391,8310
C01560=-146245,-38577,-51594,-16825,86395,8446
C01561=-146244,-38444,-53170,-16818,87391,8310
C01562=-146240,-38608,-52193,-16823,86734,8401
C01563=-146535,-35573,-50236,-16765,87015,8261
C01564=-146268,-38521,-51765,-16819,86519,8421
C01565=-147801,-39090,-52130,-16535,86146,7942
C01566=-146268,-38521,-51765,-16819,86519,8421
C01567=-144117,-44081,-61004,-17211,89666,8724
C01568=-145162,-56828,-95851,-3587,97052,36303
C01569=-147136,-55674,-91646,-3015,94990,35768
C01570=-150906,-56103,-90461,-1950,93937,34650
C01571=-150909,-57277,-89363,-1945,92659,34669
C01572=-150906,-56103,-90461,-1950,93937,34650
C01573=-147900,-55107,-89916,-2796,94193,35556
C01574=-147871,-56692,-89008,-2798,92822,35595
C01575=-149697,-57326,-89351,-2285,92656,35040
C01576=-147871,-56692,-89008,-2798,92822,35595
C01577=-149264,-52275,-86592,-2410,93564,35155
C01578=-149536,-48545,-84471,-2336,94168,35061
C01579=-149264,-52275,-86592,-2410,93564,35155
C01580=-145162,-56828,-95851,-3587,97052,36303
C01581=-148725,-41791,-46801,-46253,72923,-63254
C01582=-150766,-40622,-42529,-46203,70442,-63063
C01583=-151577,-40068,-40761,-46203,69457,-62988
C01584=-152585,-23504,-29643,-45527,70124,-63820
C01585=-151861,-23991,-31407,-45521,71087,-63922
C01586=-150038,-24992,-35653,-45558,73508,-64179
C01587=-157424,-58492,-62688,-32217,54755,-56547
C01588=-158288,-54308,-56839,-32290,53193,-56420
C01589=-158489,-51803,-54002,-32356,52725,-56354
C01590=-162920,-52118,-54243,-29783,51091,-57961
C01591=-162018,-54402,-56899,-30142,51809,-57760
C01592=-161259,-58664,-62788,-30049,53328,-57890
C01593=-162071,-38381,-52824,-22779,71448,-67723
C01594=-163630,41,-22976,-9730,99876,-85306
C01595=-164211,-2681,-21394,-9632,97468,-85315
C01596=-164465,-2984,-20111,-9597,96504,-85326
C01597=-167232,-2580,-19786,-9490,96192,-86245
C01598=-166888,-2331,-21114,-9528,97164,-86203
C01599=-166273,343,-22730,-9627,99573,-86181
C01600=-147061,-19099,-23009,-3757,61390,-3418
C01601=-130185,-5552,7433,-2044,36537,20417
C01602=-144147,-96317,-43020,16665,22045,18189
C01603=-97675,-116344,-75406,-30929,43249,-3453
C01604=-152316,-9212,-39627,-4041,74028,-36586
C01605=-151393,-4993,-15312,-4384,44467,-75506
C01606=-149831,-2435,-10935,-5835,43191,-74682
C01607=-153598,-2829,-4936,4606,33959,-78110
C01608=-153144,-5684,-1829,16153,25305,-81610
C01609=-154914,-1885,-10222,12324,42496,-79899
C01610=-154718,-4280,-13376,11999,43163,-79709
C01611=-167718,15574,1984,-24206,55458,-53961
C01612=-167855,19598,9384,-24857,53146,-53442
C01613=-167896,23400,14292,-25175,52163,-53203
C01614=-168879,23670,14551,-24625,51848,-53577
C01615=-169300,23796,14673,-24387,51714,-53738
C01616=-169985,24016,14885,-23999,51498,-54001
C01617=-170290,20267,10006,-23488,52399,-54367
C01618=-170195,16223,2573,-22831,54729,-54878
C01619=-178256,99378,67031,-19051,88552,-69176
C01620=-178526,97657,68868,-19024,86580,-68963
C01621=-177046,109131,86297,-22503,85590,-68412
C01622=-179116,103896,78898,-20485,85048,-69005
C01623=-179980,99017,72237,-18859,84943,-69225
C01624=-179276,107715,84105,-21252,84558,-69005
C01625=-180272,100173,72105,-18809,85516,-69417
C01626=-179996,101790,70145,-18825,87512,-69628
C01627=-171488,21123,-18735,-439,89529,-9365
C01628=-148539,8283,-18518,11481,74800,46031
C01629=-133884,78471,30098,11624,77529,65496
C01630=-133939,79564,34318,11736,75541,65288
C01631=-134016,73362,30598,12612,71001,64906
C01632=-130198,78667,37224,10914,68927,66030
C01633=-130560,84597,41197,10369,73487,66234
C01634=-130480,83524,36335,10225,75880,66464
C01635=-133789,96970,48697,23463,95575,62558
C01636=-133554,94997,50328,23328,93653,62262
C01637=-133529,103442,61977,22511,96128,62615
C01638=-133348,96576,53550,22948,94721,62482
C01639=-133321,94550,51417,23256,92762,62169
C01640=-128599,98999,56020,18503,91012,62952
C01641=-128273,111294,71176,17929,93549,63370
C01642=-127967,111915,71998,17889,93303,63443
C01643=-125984,92855,44553,14229,94278,63672
C01644=-118409,86943,34254,-498,98079,29639
C01645=-113225,75702,29820,-12477,90617,28537
C01646=-112952,75485,30802,-12536,89960,28691
C01647=-117762,67578,21374,-3134,88425,17539
C01648=-120996,68894,22851,4133,88343,9509
C01649=-120986,83403,30534,4203,100743,9917
C01650=-131138,87625,41047,12528,91017,-11277
C01651=-131518,88313,46232,13974,85364,-12988
C01652=-131581,87834,46842,13998,84771,-13078
C01653=-131707,87196,46726,14037,84539,-13145
C01654=-127523,76387,33616,3918,83280,-1876
C01655=-130224,83461,42270,11062,83726,-9611
C01656=-130883,82631,32190,11215,89482,-9310
C01657=-138903,29280,-14444,28707,91021,50587
C01658=-152753,-113498,-70464,41238,43505,17390
C01659=-199062,-57325,-47228,38260,64183,4080
C01660=-144700,-70309,-53328,-41384,55522,-26317
C01661=-159027,-8981,-29340,-14833,99808,-55594
C01662=-157462,-4946,-22039,-14756,97743,-54798
C01663=-155946,4301,-11330,-18807,102784,-55274
C01664=-158671,10358,-6762,-12156,106168,-56145
C01665=-156571,-6804,-23527,-14776,97863,-54502
C01666=-156840,-8773,-29171,-14894,100200,-54881
C01667=-162486,-26662,-42491,-16083,70936,-60571
C01668=-162478,-24897,-37244,-16311,68704,-60258
C01669=-161179,-32564,-36764,-20248,58009,-58071
C01670=-158579,-32364,-36623,-21541,58683,-57121
C01671=-159367,-24765,-36916,-18592,69259,-59149
C01672=-159276,-26541,-42171,-18380,71485,-59471
C01673=-144700,-70309,-53328,-41384,55522,-26317
C01674=-199062,-57325,-47228,38260,64183,4080
C01675=-152753,-113498,-70464,41238,43505,17390
C01676=-138903,29280,-14444,28707,91021,50587
C01677=-134460,43790,22046,6339,61230,73811
C01678=-133863,45767,26803,6146,59285,73930
C01679=-134509,41301,27140,7939,52069,73237
C01680=-130242,48491,34037,5055,52366,75057
C01681=-129992,52392,35365,4200,57178,75352
C01682=-129939,49644,28351,4047,60072,75482
C01683=-131463,16549,-4479,-10803,54184,75739
C01684=-132193,19548,1065,-10568,52248,75638
C01685=-132610,21611,4317,-10418,51267,75563
C01686=-134889,19383,2337,-8835,51077,74604
C01687=-134234,16346,-1785,-9163,52111,74787
C01688=-134362,13693,-7099,-8856,53981,74568
C01689=-136755,-2244,-27091,-2141,60146,66966
C01690=-152753,-113498,-70464,41238,43505,17390
C01691=-199062,-57325,-47228,38260,64183,4080
C01692=-144700,-70309,-53328,-41384,55522,-26317
C01693=-155243,-37029,-47289,-14287,81392,-50093
C01694=-162013,-14853,-33688,2862,92831,-64763
C01695=-160348,-13357,-28610,2663,90422,-64263
C01696=-158483,-5283,-21126,-235,94742,-63829
C01697=-159523,3290,-13228,4879,99055,-63648
C01698=-159523,3350,-16497,4917,101090,-63567
C01699=-158470,-14757,-33607,2451,92716,-63592
C01700=-164755,-27863,-42732,4142,59506,-66566
C01701=-162884,-23098,-35965,3113,57711,-65906
C01702=-162582,-22043,-33808,2960,56914,-65810
C01703=-159358,-22028,-33796,1037,56837,-64540
C01704=-159938,-24220,-37690,1365,58116,-64753
C01705=-160428,-28024,-42833,1630,59333,-64922
C01706=-144700,-70309,-53328,-41384,55522,-26317
C01707=-199062,-57325,-47228,38260,64183,4080
C01708=-152753,-113498,-70464,41238,43505,17390
C01709=-177120,62510,20627,9539,95868,-53949
C01710=-182918,102274,70865,2025,89904,-72285
C01711=-182573,99881,71746,1990,88125,-72198
C01712=-180645,120661,100735,-1294,86244,-71682
C01713=-175508,115553,93926,-3621,88889,-70010
C01714=-178132,93443,63515,1551,89785,-70684
C01715=-178509,95798,62536,1591,91604,-70787
C01716=-170148,25411,11260,-10861,54110,-56839
C01717=-169779,29504,18940,-11463,51585,-56403
C01718=-169637,33067,23549,-11711,50620,-56227
C01719=-164942,31927,22403,-14570,51500,-54279
C01720=-165316,28440,17904,-14160,52381,-54569
C01721=-165615,24318,10218,-13532,54869,-55036
C01722=-177120,62510,20627,9539,95868,-53949
C01723=-152753,-113498,-70464,41238,43505,17390
C01724=-199062,-57325,-47228,38260,64183,4080
C01725=-144700,-70309,-53328,-41384,55522,-26317
C01726=-142540,-54200,-62960,-20837,71495,-76935
C01727=-143745,-53250,-58469,-20670,69060,-76947
C01728=-143907,-52449,-56432,-20721,68229,-76859
C01729=-146015,-19661,-41212,-16744,94255,-78829
C01730=-145325,-27004,-46307,-16815,93781,-78527
C01731=-145058,-29561,-48130,-16841,93649,-78418
C01732=-144903,-28900,-49357,-16896,94730,-78514
C01733=-144163,-26309,-51550,-17103,97446,-78641
C01734=-174273,-50790,-66274,-423,45257,-81721
C01735=-174293,-46300,-60313,-415,43895,-81724
C01736=-174300,-44502,-57900,-412,43334,-81724
C01737=-174308,-44682,-54936,-420,41418,-81719
C01738=-174300,-46542,-57382,-423,41967,-81718
C01739=-174281,-51187,-63424,-430,43299,-81715
C01740=-170286,-21589,-54734,-4189,80944,-76248
C01741=-174005,35790,2399,-5860,112639,-83034
C01742=-174229,31517,1683,-5803,110877,-83024
C01743=-174320,29862,1474,-5782,110152,-83021
C01744=-174151,30232,3489,-5706,109139,-82910
C01745=-174234,31116,4346,-5726,109041,-82935
C01746=-174010,35219,4888,-5776,110822,-82944
C01747=-165073,-12180,-39998,-12766,95090,-81399
C01748=-146454,-66354,-59123,-37370,62542,-80053
C01749=-148014,-113391,-77231,-42747,49474,-76607
C01750=-120872,-104982,-67229,-50399,61266,-16237
C01751=-12667,-135547,-130714,31270,45596,0
BC00000=78393,670967,1075175
BC00001=177059,727519,1002542
BC00002=78393,913126,1075175
BC00003=70793,903989,1075175
BC00004=70793,903989,1075175
BC00005=70793,903989,1075175
BC00006=70793,903989,1075175
BC00007=70793,903989,1075175
BC00008=70793,903989,1075175
BC00009=70793,903989,1075175
BC00010=70793,903989,1075175
BC00011=70793,903989,1075175
BC00012=103901,897249,1075175
BC00013=103901,897249,1075175
BC00014=103901,897249,1075175
BC00015=103901,897249,1075175
BC00016=103901,897249,1075175
BC00017=103901,897249,1075175
BC00018=103901,897249,1075175
BC00019=103901,897249,1075175
BC00020=89915,910531,1075175
BC00021=89915,910531,1075175
BC00022=89915,910531,1075175
BC00023=89915,910531,1075175
BC00024=89915,910531,1075175
BC00025=89915,910531,1075175
BC00026=89915,910531,1075175
BC00027=89915,910531,1075175
BC00028=89915,910531,1075175
BC00029=27368,899646,1075175
BC00030=27368,899646,1075175
BC00031=27368,899646,1075175
BC00032=27368,899646,1075175
BC00033=27368,899646,1075175
BC00034=27368,899646,1075175
BC00035=27368,899646,1075175
BC00036=27368,899646,1075175
BC00037=160753,772187,1075175
BC00038=160753,772187,1075175
BC00039=160753,772187,1075175
BC00040=160753,772187,1075175
BC00041=160753,772187,1075175
BC00042=160753,772187,1075175
BC00043=160753,772187,1075175
BC00044=160753,772187,1075175
BC00045=160753,772187,1075175
BC00046=160753,772187,1075175
BC00047=160753,772187,1075175
BC00048=160753,772187,1075175
BC00049=123402,765716,1075175
BC00050=123402,765716,1075175
BC00051=123402,765716,1075175
BC00052=123402,765716,1075175
BC00053=123402,765716,1075175
BC00054=123402,765716,1075175
BC00055=123402,765716,1075175
BC00056=123402,765716,1075175
BC00057=123402,765716,1075175
BC00058=123402,765716,1075175
BC00059=123402,765716,1075175
BC00060=129464,768278,1075175
BC00061=151149,777443,1075175
BC00062=169689,785624,1075175
BC00063=169689,785624,1075175
BC00064=169689,785624,1075175
BC00065=169689,785624,1075175
BC00066=169689,785624,1075175
BC00067=169689,785624,1075175
BC00068=169689,785624,1075175
BC00069=169689,785624,1075175
BC00070=169689,785624,1075175
BC00071=169689,785624,1075175
BC00072=169689,785624,1075175
BC00073=169689,785624,1075175
BC00074=169689,785624,1075175
BC00075=120114,813651,1075175
BC00076=120114,813651,1075175
BC00077=120114,813651,1075175
BC00078=120114,813651,1075175
BC00079=120114,813651,1075175
BC00080=120114,813651,1075175
BC00081=120114,813651,1075175
BC00082=120114,813651,1075175
BC00083=120114,813651,1075175
BC00084=120114,813651,1075175
BC00085=120114,813651,1075175
BC00086=120114,813651,1075175
BC00087=120114,813651,1075175
BC00088=141881,838168,1075175
BC00089=141881,838168,1075175
BC00090=141881,838168,1075175
BC00091=141881,838168,1075175
BC00092=141881,838168,1075175
BC00093=141881,838168,1075175
BC00094=141881,838168,1075175
BC00095=141881,838168,1075175
BC00096=141881,838168,1075175
BC00097=141881,838168,1075175
BC00098=141881,838168,1075175
BC00099=141881,838168,1075175
BC00100=141881,838168,1075175
BC00101=69874,805894,1075175
BC00102=70019,750208,1075175
BC00103=70019,750208,1075175
BC00104=70019,750208,1075175
BC00105=70019,750208,1075175
BC00106=70019,750208,1075175
BC00107=70019,750208,1075175
BC00108=70019,750208,1075175
BC00109=70019,750208,1075175
BC00110=70019,750208,1075175
BC00111=70019,750208,1075175
BC00112=70019,750208,1075175
BC00113=70019,750208,1075175
BC00114=70019,750208,1075175
BC00115=70018,750208,1075172
BC00116=70018,750208,1075172
BC00117=70018,750208,1075172
BC00118=70018,750208,1075172
BC00119=70018,750208,1075172
BC00120=70018,750208,1075172
BC00121=70018,750208,1075172
BC00122=70018,750208,1075172
BC00123=110204,822960,1075174
BC00124=128430,855958,1075175
BC00125=125005,945340,1075175
BC00126=125005,945340,1075175
BC00127=125005,945340,1075175
BC00128=125005,945340,1075175
BC00129=125005,945340,1075175
BC00130=125005,945340,1075175
BC00131=125005,945340,1075175
BC00132=125005,945340,1075175
BC00133=125005,945340,1075175
BC00134=125005,945340,1075175
BC00135=125005,945340,1075175
BC00136=177748,940008,1075175
BC00137=177748,940008,1075175
BC00138=177748,940008,1075175
BC00139=177748,940008,1075175
BC00140=177748,940008,1075175
BC00141=177748,940008,1075175
BC00142=177748,940008,1075175
BC00143=177748,940008,1075175
BC00144=177748,940008,1075175
BC00145=177748,940008,1075175
BC00146=177748,940008,1075175
BC00147=177748,940008,1075175
BC00148=225975,953000,1075175
BC00149=225975,953000,1075175
BC00150=225975,953000,1075175
BC00151=225975,953000,1075175
BC00152=225975,953000,1075175
BC00153=225975,953000,1075175
BC00154=225975,953000,1075175
BC00155=225975,953000,1075175
BC00156=225975,953000,1075175
BC00157=225975,953000,1075175
BC00158=225975,953000,1075175
BC00159=225975,953000,1075175
BC00160=254413,953027,1075175
BC00161=252547,954523,1075175
BC00162=252548,954519,1075175
BC00163=252583,954651,1075175
BC00164=252019,957675,1075175
BC00165=252583,954651,1075175
BC00166=252165,954787,1075175
BC00167=249030,954243,1075175
BC00168=252165,954787,1075175
BC00169=258696,949550,1075175
BC00170=251448,951648,1075175
BC00171=250551,956448,1075175
BC00172=250192,958368,1075175
BC00173=250193,958364,1075175
BC00174=250073,958395,1075175
BC00175=249509,961419,1075175
BC00176=250073,958395,1075175
BC00177=251329,951675,1075175
BC00178=248439,993035,1075175
BC00179=271638,1017285,1075175
BC00180=314947,1062557,1075175
BC00181=311280,1056373,1075175
BC00182=310409,1054905,1075175
BC00183=310409,1054901,1075175
BC00184=310409,1054905,1075175
BC00185=284329,1066137,1075175
BC00186=285931,1063482,1075175
BC00187=284329,1066137,1075175
BC00188=333588,1039325,1075175
BC00189=330835,1037779,1075175
BC00190=333588,1039325,1075175
BC00191=340460,1045393,1075175
BC00192=296133,1047687,1075175
BC00193=279319,1048558,1075175
BC00194=281895,1044284,1075175
BC00195=282926,1042574,1075175
BC00196=282926,1042570,1075175
BC00197=282744,1042486,1075175
BC00198=284346,1039831,1075175
BC00199=282744,1042486,1075175
BC00200=279137,1048470,1075175
BC00201=253507,1028204,1074244
BC00202=212842,1022781,1075175
BC00203=146334,1015862,1075175
BC00204=66205,1045023,1075175
BC00205=66205,1045023,1075175
BC00206=66205,1045023,1075175
BC00207=66205,1045023,1075175
BC00208=66205,1045023,1075175
BC00209=66205,1045023,1075175
BC00210=66205,1045023,1075175
BC00211=66205,1045023,1075175
BC00212=66205,1045023,1075175
BC00213=66205,1045023,1075175
BC00214=66205,1045023,1075175
BC00215=66205,1045023,1075175
BC00216=125029,959783,1075175
BC00217=190390,972133,1075175
BC00218=190390,972133,1075175
BC00219=190390,972133,1075173
BC00220=190390,972133,1075175
BC00221=190390,972133,1075175
BC00222=190390,972133,1075175
BC00223=190390,972133,1075175
BC00224=190390,972133,1075175
BC00225=190390,972133,1075175
BC00226=190390,972133,1075175
BC00227=190390,972133,1075175
BC00228=190390,972133,1075175
BC00229=190390,972133,1075175
BC00230=103363,888035,1075175
BC00231=35304,822265,1075175
BC00232=35304,822265,1075175
BC00233=35304,822265,1075175
BC00234=35304,822265,1075175
BC00235=35304,822265,1075175
BC00236=35304,822265,1075175
BC00237=35304,822265,1075175
BC00238=35304,822265,1075175
BC00239=35304,822265,1075175
BC00240=35304,822265,1075175
BC00241=35304,822265,1075175
BC00242=35304,822265,1075175
BC00243=167967,799945,1075175
BC00244=311305,898961,1075175
BC00245=311305,898961,1075175
BC00246=311305,898961,1075175
BC00247=311305,898961,1075175
BC00248=311305,898961,1075175
BC00249=311305,898961,1075175
BC00250=311305,898961,1075175
BC00251=311305,898961,1075175
BC00252=311305,898961,1075175
BC00253=311305,898961,1075175
BC00254=311305,898961,1075175
BC00255=311305,898961,1075175
BC00256=113180,824290,1075229
BC00257=113180,824290,1075229
BC00258=113180,824290,1075229
BC00259=113180,824290,1075229
BC00260=113180,824290,1075229
BC00261=113180,824290,1075229
BC00262=113180,824290,1075229
BC00263=113180,824290,1075229
BC00264=113180,824290,1075229
BC00265=113180,824290,1075229
BC00266=113180,824290,1075229
BC00267=113180,824290,1075229
BC00268=355762,967535,1075175
BC00269=355762,967535,1075175
BC00270=355762,967535,1075175
BC00271=355762,967535,1075175
BC00272=355762,967535,1075175
BC00273=355762,967535,1075175
BC00274=355762,967535,1075175
BC00275=355762,967535,1075175
BC00276=397203,974799,1075175
BC00277=397203,974799,1075175
BC00278=397203,974799,1075175
BC00279=397203,974799,1075175
BC00280=397203,974799,1075175
BC00281=397203,974799,1075175
BC00282=397203,974799,1075175
BC00283=397203,974799,1075175
BC00284=279782,952911,1075175
BC00285=264332,967435,1075175
BC00286=264332,967435,1075175
BC00287=264332,967435,1075175
BC00288=264332,967435,1075175
BC00289=264332,967435,1075175
BC00290=264332,967435,1075175
BC00291=264332,967435,1075175
BC00292=264332,967435,1075175
BC00293=264332,967435,1075175
BC00294=264332,967435,1075175
BC00295=264332,967435,1075175
BC00296=290594,956201,1075175
BC00297=316856,944967,1075175
BC00298=316856,944967,1075175
BC00299=316856,944967,1075175
BC00300=316856,944967,1075175
BC00301=316856,944967,1075175
BC00302=316856,944967,1075175
BC00303=316856,944967,1075175
BC00304=316856,944967,1075175
BC00305=316856,944967,1075175
BC00306=316856,944967,1075175
BC00307=316856,944967,1075175
BC00308=316856,944967,1075175
BC00309=316856,944967,1075175
BC00310=316856,944967,1075175
BC00311=316856,944967,1075175
BC00312=316856,944967,1075175
BC00313=329946,891084,1075175
BC00314=337525,859888,1075175
BC00315=337525,859888,1075175
BC00316=337525,859888,1075175
BC00317=337525,859888,1075175
BC00318=337525,859888,1075175
BC00319=337525,859888,1075175
BC00320=337525,859888,1075175
BC00321=337525,859888,1075175
BC00322=238148,874377,1075175
BC00323=227206,875826,1075175
BC00324=227206,875826,1075175
BC00325=227206,875826,1075175
BC00326=227206,875826,1075175
BC00327=227206,875826,1075175
BC00328=227206,875826,1075175
BC00329=280946,887675,1075175
BC00330=280946,887675,1075175
BC00331=280946,887675,1075175
BC00332=280946,887675,1075175
BC00333=280946,887675,1075175
BC00334=280946,887675,1075175
BC00335=280946,887675,1075175
BC00336=280946,887675,1075175
BC00337=239261,850045,1075175
BC00338=207869,857354,1075175
BC00339=207869,857354,1075175
BC00340=207869,857354,1075175
BC00341=207869,857354,1075175
BC00342=207869,857354,1075175
BC00343=207869,857354,1075175
BC00344=207869,857354,1075175
BC00345=207869,857354,1075175
BC00346=207996,857850,1075175
BC00347=184532,936508,1075175
BC00348=163675,1006427,1075175
BC00349=164114,1001741,1075175
BC00350=164289,999867,1075175
BC00351=160191,997498,1075175
BC00352=158450,996490,1075175
BC00353=154353,994119,1075175
BC00354=154178,995993,1075175
BC00355=153739,1000679,1075175
BC00356=82719,974634,1075175
BC00357=82719,974634,1075175
BC00358=82720,974634,1075172
BC00359=82720,974634,1075172
BC00360=82719,974634,1075175
BC00361=82720,974634,1075173
BC00362=82719,974634,1075175
BC00363=82719,974634,1075175
BC00364=70441,948911,1075175
BC00365=70441,948911,1075175
BC00366=70441,948911,1075175
BC00367=70441,948911,1075175
BC00368=70441,948911,1075175
BC00369=70441,948911,1075175
BC00370=182218,957850,1075175
BC00371=274997,1000420,1075175
BC00372=293323,1008828,1075175
BC00373=293323,1008828,1075175
BC00374=293323,1008828,1075175
BC00375=293323,1008828,1075175
BC00376=293323,1008828,1075175
BC00377=293323,1008828,1075175
BC00378=337244,1059629,1075175
BC00379=337244,1059629,1075175
BC00380=337244,1059629,1075175
BC00381=337244,1059629,1075175
BC00382=337244,1059629,1075175
BC00383=337244,1059629,1075175
BC00384=337244,1059629,1075175
BC00385=227430,982125,1075175
BC00386=115014,939685,1075175
BC00387=118867,937244,1075175
BC00388=120408,936268,1075175
BC00389=140995,947826,1075175
BC00390=182041,976368,1075175
BC00391=180846,977671,1075175
BC00392=177859,980929,1075175
BC00393=194800,984537,1075175
BC00394=244653,1016084,1075175
BC00395=241511,1010564,1075175
BC00396=240254,1008357,1075175
BC00397=240254,1008354,1075175
BC00398=241511,1010562,1075175
BC00399=244653,1016081,1075175
BC00400=244653,1016084,1075175
BC00401=272695,1033702,1075175
BC00402=285514,1041756,1075175
BC00403=284751,1045931,1075175
BC00404=282162,1039999,1075175
BC00405=281126,1037626,1075175
BC00406=207140,1028015,1075175
BC00407=260829,1058016,1075175
BC00408=212034,1012943,1075175
BC00409=209227,1012918,1075175
BC00410=202210,1012854,1075175
BC00411=196613,982513,1075175
BC00412=175963,870568,1075175
BC00413=163612,803610,1075175
BC00414=152631,778532,1075175
BC00415=146092,780306,1075175
BC00416=143477,781016,1075175
BC00417=143597,781078,1075175
BC00418=143625,781092,1075175
BC00419=143746,781156,1075175
BC00420=146361,780446,1075175
BC00421=152900,778672,1075175
BC00422=152900,778672,1075175
BC00423=74084,744686,1075175
BC00424=74084,744686,1075175
BC00425=67287,679894,1075175
BC00426=67287,679894,1075175
BC00427=67287,679894,1075175
BC00428=67287,679894,1075175
BC00429=67287,679894,1075175
BC00430=67287,679894,1075175
BC00431=67287,679894,1075175
BC00432=67287,679894,1075175
BC00433=83395,694294,1075175
BC00434=102108,711022,1075175
BC00435=165558,767742,1075175
BC00436=222482,818628,1075175
BC00437=215814,820321,1075175
BC00438=213147,820999,1075175
BC00439=213147,820994,1075175
BC00440=213147,820993,1075175
BC00441=213148,820988,1075175
BC00442=215815,820311,1075175
BC00443=222483,818617,1075175
BC00444=173722,816110,1075175
BC00445=90356,811823,1075175
BC00446=89696,811574,1075175
BC00447=89432,811475,1075175
BC00448=85301,809160,1075175
BC00449=73323,802435,1075175
BC00450=69196,800114,1075175
BC00451=69460,800213,1075175
BC00452=70120,800462,1075175
BC00453=203969,867991,1075175
BC00454=200192,866637,1075175
BC00455=198681,866095,1075175
BC00456=196278,870078,1075175
BC00457=188025,883752,1075175
BC00458=185620,887734,1075175
BC00459=187131,888276,1075175
BC00460=190907,889630,1075175
BC00461=185807,834457,1075175
BC00462=185042,826181,1075175
BC00463=182820,831186,1075175
BC00464=181931,833188,1075175
BC00465=205283,846231,1075175
BC00466=246906,863634,1075175
BC00467=246906,863634,1075175
BC00468=248214,861732,1075175
BC00469=251484,856977,1075175
BC00470=177002,833071,1075175
BC00471=153563,828435,1075175
